// TIA Portal V20 export
// export: Created 2025-12-01T14:56:37.1159273Z, ExportSetting None, DisplayName Totally Integrated Automation Portal, DisplayVersion V20 Update 3, DisplayName TIA Portal Openness, DisplayVersion V20 Update 3, DisplayName TIA Portal Version Control Interface, DisplayVersion V20 Update 3, DisplayName STEP 7 Professional, DisplayVersion V20 Update 3, DisplayName STEP 7 Safety, DisplayVersion V20 Update 2, DisplayName WinCC Basic/Comfort/Advanced, DisplayVersion V20 Update 3, DisplayName WinCC Professional, DisplayVersion V20 Update 3, DisplayName WinCC Unified, DisplayVersion V20 Update 3
FUNCTION_BLOCK "FB12_M_PASO_ELEV_E1E2E3E4_S1S2S3S4_UPDW"   // FB12, LAD
TITLE = Control del Ramal de Salidas
{ S7_Optimized_Access := 'FALSE' }
AUTHOR : M_ELEVA
NAME : 20160509
VERSION : 3.7
// stored: AutoNumber false, SetENOAutomatically false
   VAR_INPUT
      Mesa : UInt;   // Mesa de la FB
      Error_Tx : Bool;   // Error en el Tx
      EnTension : Bool;   // Existe Tension en la Mesa
      Termico_Tx : Bool;   // Proteccion del Tx
      pHsMx_1 : Bool;   // pHs de la Mesa (Para Entrada por E3E4)
      pHsMx_2 : Bool;   // pHs de la Mesa (Para Entrada por E1E2)
      pHsMx_PR1 : Bool;   // pHs de Protrusion de la Mesa. Nota: No existe >> ON
      pHsMx_PR3 : Bool;   // pHs de Protrusion de la Mesa. Nota: No existe >> ON
      Avance_Tx : Bool;   // Avance del Tx
      Retroceso_Tx : Bool;   // Retroceso del Tx
      Termico_MELEV : Bool;   // Protecion de la Mesa Elevadora
      MELEV_DetectorSeg : Bool;   // Detector de Seguridad >>> Mesa Elevadora
      MELEV_UP : Bool;   // Posicion Arriba >>> Mesa Elevadora
      MELEV_DW : Bool;   // Posicion Abajo >>> Mesa Elevadora
      MELEV_EnMovimiento : Bool;   // EnMovimiento >>> Mesa Elevadora
      Pos_Rep_Vacio_DW : Bool;   // Pos. Reposo Vacia DW >>> Config
      Pos_Rep_Vacio_UP : Bool;   // Pos. Reposo Vacia UP >>> Config
      Pos_Rep_Carga_DW : Bool;   // Pos. Reposo Cargada DW >>> Config
      Pos_Rep_Carga_UP : Bool;   // Pos. Reposo Cargada UP >>> Config
      MAnt_DescargaAct_M1_DW : Bool;   // E1 >> Mesa Anterior DescargaAct
      AVTF_Ent_M1_DW : Bool;   // E1 >> Mesa Anterior AVTF
      P_Mens_Ent_M1_DW : Bool;   // E1 >> Mesa Anterior P_Mens
      MAnt_DescargaAct_M3_DW : Bool;   // E3 >> Mesa Anterior DescargaAct
      AVTF_Ent_M3_DW : Bool;   // E3 >> Mesa Anterior AVTF
      P_Mens_Ent_M3_DW : Bool;   // E3 >> Mesa Anterior P_Mens
      PTF_Sal_M1_DW : Bool;   // S1 >> Mesa Siguiente PTF
      FTF_Sal_M1_DW : Bool;   // S1 >> Mesa Siguiente FTF
      PTF_Sal_M3_DW : Bool;   // S3 >> Mesa Siguiente PTF
      FTF_Sal_M3_DW : Bool;   // S3 >> Mesa Siguiente FTF
      MSig_CargaAct_M1_DW : Bool;
      MSig_CargaAct_M3_DW : Bool;
      MAnt_DescargaAct_M2_UP : Bool;   // E2 >> Mesa Anterior DescargaAct
      AVF_Ent_M2_UP : Bool;   // E2 >> Mesa Anterior AVTF
      P_Mens_Ent_M2_UP : Bool;   // E2 >> Mesa Anterior P_Mens
      MAnt_DescargaAct_M4_UP : Bool;   // E4 >> Mesa Anterior DescargaAct
      AVTF_Ent_M4_UP : Bool;   // E4 >> Mesa Anterior AVTF
      P_Mens_Ent_M4_UP : Bool;   // E4 >> Mesa Anterior P_Mens
      PTF_Sal_M2_UP : Bool;   // S2 >> Mesa Siguiente PTF
      FTF_Sal_M2_UP : Bool;   // S2 >> Mesa Siguiente FTF
      PTF_Sal_M4_UP : Bool;   // S4 >> Mesa Siguiente PTF
      FTF_Sal_M4_UP : Bool;   // S4 >> Mesa Siguiente FTF
      MSig_CargaAct_M2_UP : Bool;
      MSig_CargaAct_M4_UP : Bool;
      Mx_VelocidadLenta_In : Bool;   // Forzar a Velociada Lenta
      F_ENV_MENS_Mx : Bool;   // Fin de Envio de Mensaje
      OrdSal_M1_DW : Bool;   // Orden de Salida por S1
      OrdSal_M3_DW : Bool;   // Orden de Salida por S3
      OrdSal_M2_UP : Bool;   // Orden de Salida por S2
      OrdSal_M4_UP : Bool;   // Orden de Salida por S4
      V_CNT_pHsMx : Int := 1000;   // Valor de Presencia
      V_CNT_pHsMx_FTF : Int := 200;   // Valor para activar FTF. Nota: < = V_CNT_pHsMx.
      V_CNTSeg_pHsMx : Int := 2000;   // Valor de Seguriadad para Presencia
      V_CNT_PasoLenta : Int := 2000;   // Valor de Paso a Lenta
      V_CNT_ApHsMx : Int := 200;   // Valor de Ausencia
      V_CNTSeg_ApHsMx : Int := 2000;   // Valor de Seguriadad para Ausencia
      V_TOut_Tx_Mx : Int := 30000;   // TimeOut de Entrada por E1
      V_TOut_MELEV : Int := 5000;   // TimeOut de Mesa Elevadora
      V_TMP_Protrusion : Int := 200;   // TMP de Protrusion
      V_CNT_PerdidapHs : Int := 1000;   // CNT de Perdida de pHs
   END_VAR
   VAR_OUTPUT
      P_EnvMens_PMx : Bool;   // Permiso de Enviar Mensaje de Presencia
      P_RecepOK_Mx : Bool;   // Recepcion OK
      PTF_Ent_M1_DW : Bool;   // E1 >> Mesa Anterior PTF
      FTF_Ent_M1_DW : Bool;   // E1 >> Mesa Anterior FTF
      PTF_Ent_M3_DW : Bool;   // E3 >> Mesa Anterior PTF
      FTF_Ent_M3_DW : Bool;   // E3 >> Mesa Anterior FTF
      AVTF_Sal_M1_DW : Bool;   // S1 >> Mesa Siguiente AVTF
      P_Mens_Sal_M1_DW : Bool;   // S1 >> Mesa Siguiente P_Mens
      AVTF_Sal_M3_DW : Bool;   // S3 >> Mesa Siguiente AVTF
      P_Mens_Sal_M3_DW : Bool;   // S3 >> Mesa Siguiente P_Mens
      PTF_Ent_M2_UP : Bool;   // E2 >> Mesa Anterior PTF
      FTF_Ent_M2_UP : Bool;   // E2 >> Mesa Anterior FTF
      PTF_Ent_M4_UP : Bool;   // E4 >> Mesa Anterior PTF
      FTF_Ent_M4_UP : Bool;   // E4 >> Mesa Anterior FTF
      AVTF_Sal_M2_UP : Bool;   // S2 >> Mesa Siguiente AVTF
      P_Mens_Sal_M2_UP : Bool;   // S2 >> Mesa Siguiente P_Mens
      AVTF_Sal_M4_UP : Bool;   // S4 >> Mesa Siguiente AVTF
      P_Mens_Sal_M4_UP : Bool;   // S4 >> Mesa Siguiente P_Mens
   END_VAR
   VAR
      Anular_pr1 : Bool;   // ???
      Anular_pr3 : Bool;   // ???
      Mx_ET00 : Bool;
      Mx_ET01 { ExternalWritable := 'False'} : Bool;
      Mx_ET02 : Bool;
      Mx_ET08 : Bool;
      Mx_ET09 : Bool;
      Mx_ET10 : Bool;
      Mx_ET11 : Bool;
      Mx_ET12 : Bool;
      Mx_ET110 : Bool;
      Mx_ET111 : Bool;
      Mx_ET50 : Bool;
      Mx_ET51 : Bool;
      Mx_ET150 : Bool;
      Mx_ET151 : Bool;
      Selec_UP : Bool;   // Seleccionado UP de la Mesa Elevadora
      Selec_DW : Bool;   // Seleccionado DW de la Mesa Elevadora
      Selec_M1M2_Entrada : Bool;   // Seleccionado Entrada E1_DW y E2_UP
      Selec_M3M4_Entrada : Bool;   // Seleccionado Entrada E3_DW y E4_UP
      Selec_M1M2_Salida : Bool;   // Seleccionado Salida E1_DW y E2_UP
      Selec_M3M4_Salida : Bool;   // Seleccionado Salida E3_DW y E4_UP
      MEnt_DescargaAct : Bool;   // Interlock >> DesCargaAct de MAnt >> Mx
      AVTF_MEnt : Bool;   // Interlock >> AVTF de MAnt >> Mx
      P_Mens_MEnt : Bool;   // Interlock >> P_Mens de MAnt >> Mx
      PTF_MEnt : Bool;   // Interlock >> PTF de MAnt >> Mx
      FTF_MEnt : Bool;   // Interlock >> FTF de MAnt >> Mx
      AVTF_MSal : Bool;   // Interlock >> AVTF de Mx >> MSig
      P_Mens_MSal : Bool;   // Interlock >> P_Mens de Mx >> MSig
      PTF_MSal : Bool;   // Interlock >> PTF de Mx >> MSig
      FTF_MSal : Bool;   // Interlock >> FTF de Mx >> MSig
      ProtocoloInciado : Bool;   // Iniciado el Envio del Mensaje de Presencia
      STAT_EnvMens_PMx : Bool;   // Interna >> Envio del Mensaje de Presencia
      CNT_pHsMx_FTF_OK : Bool;   // Enviar ya FTF
      CNT_pHsMx { S7_SetPoint := 'True'} : "FB910_CNT_UHS";   // CNT de la Presencia
      CNTSeg_pHsMx { S7_SetPoint := 'True'} : "FB910_CNT_UHS";   // CNT de Seguridad de la Presencia
      CNT_ApHsMx { S7_SetPoint := 'True'} : "FB910_CNT_UHS";   // CNT de la Ausencia
      CNTSeg_ApHsMx { S7_SetPoint := 'True'} : "FB910_CNT_UHS";   // CNT de Seguridad de la Ausencia
      TMP_EnTension { S7_SetPoint := 'True'} : "FB910_CNT_UHS";
      TOut_Av_Mx { S7_SetPoint := 'True'} : "FB910_CNT_UHS";   // Time Out de Entrada de E1 o E2
      TOut_Rt_Mx { S7_SetPoint := 'True'} : "FB910_CNT_UHS";   // Time Out de Entrada de E3 o E4
      TOut_Subir_MELEV { S7_SetPoint := 'True'} : "FB910_CNT_UHS";   // Time Out de Subida de Mesa Elevadora
      TOut_Bajar_MELEV { S7_SetPoint := 'True'} : "FB910_CNT_UHS";   // Time Out de Bajada de Mesa Elevadora
      TMP_Protrusion { S7_SetPoint := 'True'} : "FB910_CNT_UHS";   // TMP de la Protrusion
      CNT_PerdidapHs { S7_SetPoint := 'True'} : "FB910_CNT_UHS";   // CNT de Perdida de pHs
   END_VAR
   VAR_TEMP
      EstadoZona : "EstadoZona";   // Estado de Zona de la Mesa
      EstadoVI : "EstadosMesa";   // Estado del Vehiculo Inteliguente de la Mesa
      ConfigFB : "UDT_ConfigFB";   // Configuracion de la FB de la Mesa
      V_Protrusion : Int;
      Aux_ET00 : Bool;
   END_VAR
   VAR_TEMP   // added for the SCL form of the ladder/FBD networks
      _w1 : Bool;
      _w2 : Bool;
      _w3 : Bool;
      _w4 : Bool;
      _w5 : Bool;
      _w6 : Bool;
   END_VAR
BEGIN

REGION Network 1: INICIALIZAR - Recoger las Variables de Estado de la Mesa
   // Se recoge - Estado_CBx
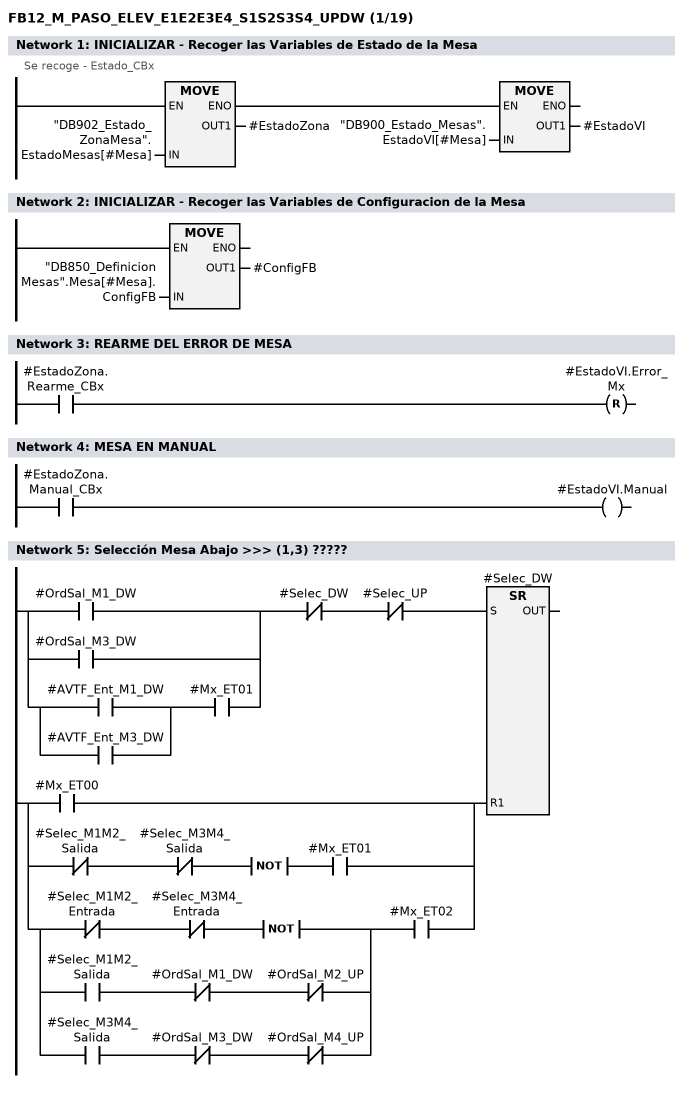
   RUNG wire#powerrail
      Move(in := "DB902_Estado_ZonaMesa".EstadoMesas[#Mesa], out1 => #EstadoZona)
      Move(in := "DB900_Estado_Mesas".EstadoVI[#Mesa], out1 => #EstadoVI)
   END_RUNG
   // the same network as SCL:
   #EstadoZona := "DB902_Estado_ZonaMesa".EstadoMesas[#Mesa];
   #EstadoVI := "DB900_Estado_Mesas".EstadoVI[#Mesa];
END_REGION

REGION Network 2: INICIALIZAR - Recoger las Variables de Configuracion de la Mesa
   RUNG wire#powerrail
      Move(in := "DB850_DefinicionMesas".Mesa[#Mesa].ConfigFB, out1 => #ConfigFB)
   END_RUNG
   // the same network as SCL:
   #ConfigFB := "DB850_DefinicionMesas".Mesa[#Mesa].ConfigFB;
END_REGION

REGION Network 3: REARME DEL ERROR DE MESA
   RUNG wire#powerrail
      Contact( #EstadoZona.Rearme_CBx )
      R_Coil( #EstadoVI.Error_Mx )
   END_RUNG
   // the same network as SCL:
   IF #EstadoZona.Rearme_CBx THEN #EstadoVI.Error_Mx := FALSE; END_IF;
END_REGION

REGION Network 4: MESA EN MANUAL
   RUNG wire#powerrail
      Contact( #EstadoZona.Manual_CBx )
      Coil( #EstadoVI.Manual )
   END_RUNG
   // the same network as SCL:
   #EstadoVI.Manual := #EstadoZona.Manual_CBx;
END_REGION

REGION Network 5: Selección Mesa Abajo >>> (1,3) ?????
   RUNG wire#powerrail
      Contact( #OrdSal_M1_DW )
      wire#w1
      I_Contact( #Selec_DW )
      I_Contact( #Selec_UP )
      S_SR(operand := #Selec_DW, r1 := wire#w4)
   END_RUNG
   RUNG wire#powerrail
      Contact( #OrdSal_M3_DW )
   END_RUNG wire#w1
   RUNG wire#powerrail
      Contact( #AVTF_Ent_M1_DW )
      wire#w2
      Contact( #Mx_ET01 )
   END_RUNG wire#w1
   RUNG wire#powerrail
      Contact( #AVTF_Ent_M3_DW )
   END_RUNG wire#w2
   RUNG wire#powerrail
      Contact( #Mx_ET00 )
   END_RUNG wire#w4
   RUNG wire#powerrail
      I_Contact( #Selec_M1M2_Salida )
      I_Contact( #Selec_M3M4_Salida )
      Not()
      Contact( #Mx_ET01 )
   END_RUNG wire#w4
   RUNG wire#powerrail
      I_Contact( #Selec_M1M2_Entrada )
      I_Contact( #Selec_M3M4_Entrada )
      Not()
      wire#w3
      Contact( #Mx_ET02 )
   END_RUNG wire#w4
   RUNG wire#powerrail
      Contact( #Selec_M1M2_Salida )
      I_Contact( #OrdSal_M1_DW )
      I_Contact( #OrdSal_M2_UP )
   END_RUNG wire#w3
   RUNG wire#powerrail
      Contact( #Selec_M3M4_Salida )
      I_Contact( #OrdSal_M3_DW )
      I_Contact( #OrdSal_M4_UP )
   END_RUNG wire#w3
   // the same network as SCL:
   IF (#OrdSal_M1_DW OR #OrdSal_M3_DW OR ((#AVTF_Ent_M1_DW OR #AVTF_Ent_M3_DW) AND #Mx_ET01)) AND NOT #Selec_DW AND NOT #Selec_UP THEN
       #Selec_DW := TRUE;   // SR flip-flop
   END_IF;
   IF #Mx_ET00 OR (NOT (NOT #Selec_M1M2_Salida AND NOT #Selec_M3M4_Salida) AND #Mx_ET01) OR ((NOT (NOT #Selec_M1M2_Entrada AND NOT #Selec_M3M4_Entrada) OR (#Selec_M1M2_Salida AND NOT #OrdSal_M1_DW AND NOT #OrdSal_M2_UP) OR (#Selec_M3M4_Salida AND NOT #OrdSal_M3_DW AND NOT #OrdSal_M4_UP)) AND #Mx_ET02) THEN
       #Selec_DW := FALSE;
   END_IF;
END_REGION

REGION Network 6: Selección Mesa Arriba >>> (2,4) ?????
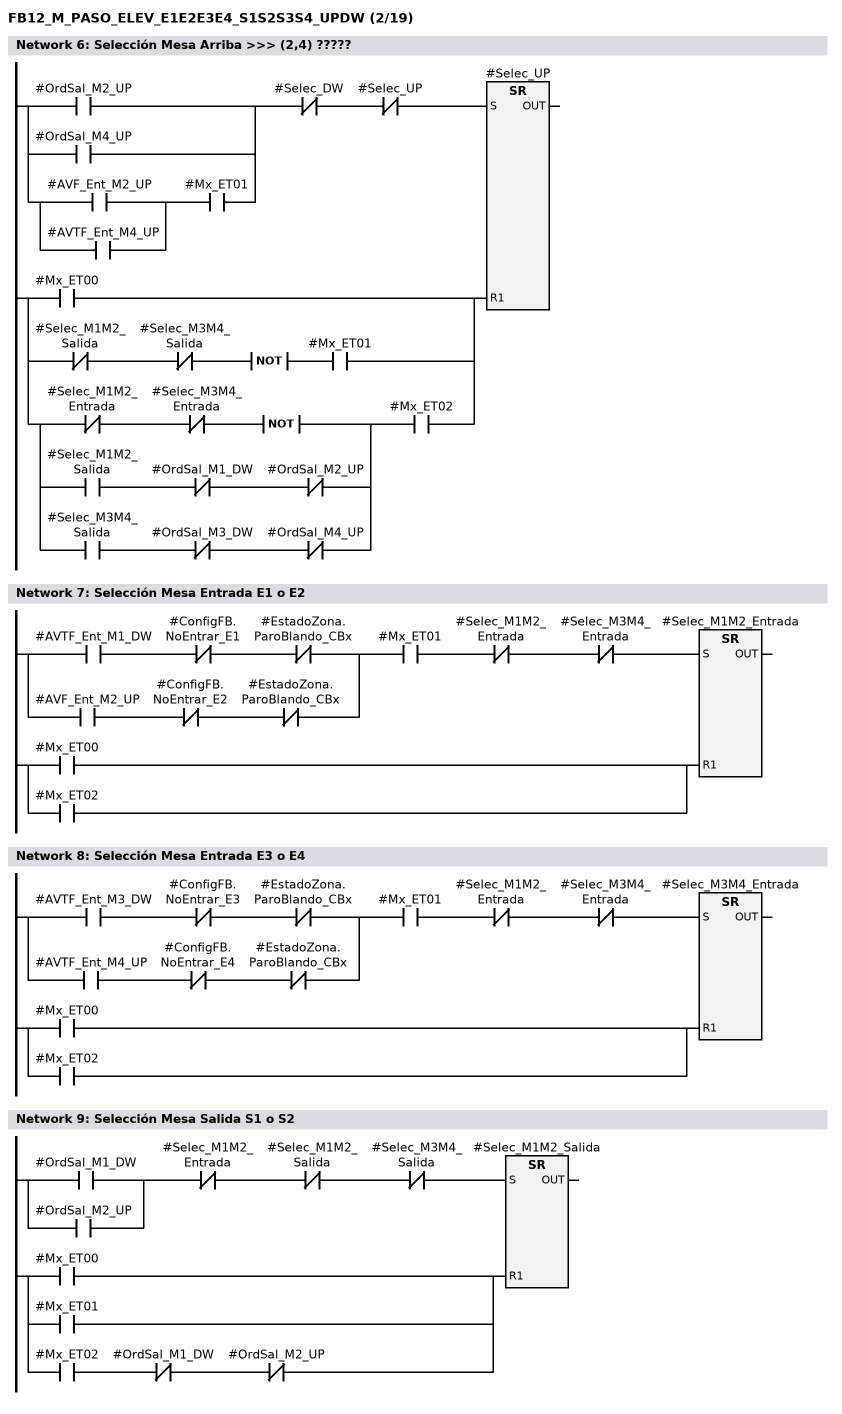
   RUNG wire#powerrail
      Contact( #OrdSal_M2_UP )
      wire#w1
      I_Contact( #Selec_DW )
      I_Contact( #Selec_UP )
      S_SR(operand := #Selec_UP, r1 := wire#w4)
   END_RUNG
   RUNG wire#powerrail
      Contact( #OrdSal_M4_UP )
   END_RUNG wire#w1
   RUNG wire#powerrail
      Contact( #AVF_Ent_M2_UP )
      wire#w2
      Contact( #Mx_ET01 )
   END_RUNG wire#w1
   RUNG wire#powerrail
      Contact( #AVTF_Ent_M4_UP )
   END_RUNG wire#w2
   RUNG wire#powerrail
      Contact( #Mx_ET00 )
   END_RUNG wire#w4
   RUNG wire#powerrail
      I_Contact( #Selec_M1M2_Salida )
      I_Contact( #Selec_M3M4_Salida )
      Not()
      Contact( #Mx_ET01 )
   END_RUNG wire#w4
   RUNG wire#powerrail
      I_Contact( #Selec_M1M2_Entrada )
      I_Contact( #Selec_M3M4_Entrada )
      Not()
      wire#w3
      Contact( #Mx_ET02 )
   END_RUNG wire#w4
   RUNG wire#powerrail
      Contact( #Selec_M1M2_Salida )
      I_Contact( #OrdSal_M1_DW )
      I_Contact( #OrdSal_M2_UP )
   END_RUNG wire#w3
   RUNG wire#powerrail
      Contact( #Selec_M3M4_Salida )
      I_Contact( #OrdSal_M3_DW )
      I_Contact( #OrdSal_M4_UP )
   END_RUNG wire#w3
   // the same network as SCL:
   IF (#OrdSal_M2_UP OR #OrdSal_M4_UP OR ((#AVF_Ent_M2_UP OR #AVTF_Ent_M4_UP) AND #Mx_ET01)) AND NOT #Selec_DW AND NOT #Selec_UP THEN
       #Selec_UP := TRUE;   // SR flip-flop
   END_IF;
   IF #Mx_ET00 OR (NOT (NOT #Selec_M1M2_Salida AND NOT #Selec_M3M4_Salida) AND #Mx_ET01) OR ((NOT (NOT #Selec_M1M2_Entrada AND NOT #Selec_M3M4_Entrada) OR (#Selec_M1M2_Salida AND NOT #OrdSal_M1_DW AND NOT #OrdSal_M2_UP) OR (#Selec_M3M4_Salida AND NOT #OrdSal_M3_DW AND NOT #OrdSal_M4_UP)) AND #Mx_ET02) THEN
       #Selec_UP := FALSE;
   END_IF;
END_REGION

REGION Network 7: Selección Mesa Entrada E1 o E2
   RUNG wire#powerrail
      Contact( #AVTF_Ent_M1_DW )
      I_Contact( #ConfigFB.NoEntrar_E1 )
      I_Contact( #EstadoZona.ParoBlando_CBx )
      wire#w1
      Contact( #Mx_ET01 )
      I_Contact( #Selec_M1M2_Entrada )
      I_Contact( #Selec_M3M4_Entrada )
      S_SR(operand := #Selec_M1M2_Entrada, r1 := wire#w2)
   END_RUNG
   RUNG wire#powerrail
      Contact( #AVF_Ent_M2_UP )
      I_Contact( #ConfigFB.NoEntrar_E2 )
      I_Contact( #EstadoZona.ParoBlando_CBx )
   END_RUNG wire#w1
   RUNG wire#powerrail
      Contact( #Mx_ET00 )
   END_RUNG wire#w2
   RUNG wire#powerrail
      Contact( #Mx_ET02 )
   END_RUNG wire#w2
   // the same network as SCL:
   IF ((#AVTF_Ent_M1_DW AND NOT #ConfigFB.NoEntrar_E1 AND NOT #EstadoZona.ParoBlando_CBx) OR (#AVF_Ent_M2_UP AND NOT #ConfigFB.NoEntrar_E2 AND NOT #EstadoZona.ParoBlando_CBx)) AND #Mx_ET01 AND NOT #Selec_M1M2_Entrada AND NOT #Selec_M3M4_Entrada THEN
       #Selec_M1M2_Entrada := TRUE;   // SR flip-flop
   END_IF;
   IF #Mx_ET00 OR #Mx_ET02 THEN #Selec_M1M2_Entrada := FALSE; END_IF;
END_REGION

REGION Network 8: Selección Mesa Entrada E3 o E4
   RUNG wire#powerrail
      Contact( #AVTF_Ent_M3_DW )
      I_Contact( #ConfigFB.NoEntrar_E3 )
      I_Contact( #EstadoZona.ParoBlando_CBx )
      wire#w1
      Contact( #Mx_ET01 )
      I_Contact( #Selec_M1M2_Entrada )
      I_Contact( #Selec_M3M4_Entrada )
      S_SR(operand := #Selec_M3M4_Entrada, r1 := wire#w2)
   END_RUNG
   RUNG wire#powerrail
      Contact( #AVTF_Ent_M4_UP )
      I_Contact( #ConfigFB.NoEntrar_E4 )
      I_Contact( #EstadoZona.ParoBlando_CBx )
   END_RUNG wire#w1
   RUNG wire#powerrail
      Contact( #Mx_ET00 )
   END_RUNG wire#w2
   RUNG wire#powerrail
      Contact( #Mx_ET02 )
   END_RUNG wire#w2
   // the same network as SCL:
   IF ((#AVTF_Ent_M3_DW AND NOT #ConfigFB.NoEntrar_E3 AND NOT #EstadoZona.ParoBlando_CBx) OR (#AVTF_Ent_M4_UP AND NOT #ConfigFB.NoEntrar_E4 AND NOT #EstadoZona.ParoBlando_CBx)) AND #Mx_ET01 AND NOT #Selec_M1M2_Entrada AND NOT #Selec_M3M4_Entrada THEN
       #Selec_M3M4_Entrada := TRUE;   // SR flip-flop
   END_IF;
   IF #Mx_ET00 OR #Mx_ET02 THEN #Selec_M3M4_Entrada := FALSE; END_IF;
END_REGION

REGION Network 9: Selección Mesa Salida S1 o S2
   RUNG wire#powerrail
      Contact( #OrdSal_M1_DW )
      wire#w1
      I_Contact( #Selec_M1M2_Entrada )
      I_Contact( #Selec_M1M2_Salida )
      I_Contact( #Selec_M3M4_Salida )
      S_SR(operand := #Selec_M1M2_Salida, r1 := wire#w2)
   END_RUNG
   RUNG wire#powerrail
      Contact( #OrdSal_M2_UP )
   END_RUNG wire#w1
   RUNG wire#powerrail
      Contact( #Mx_ET00 )
   END_RUNG wire#w2
   RUNG wire#powerrail
      Contact( #Mx_ET01 )
   END_RUNG wire#w2
   RUNG wire#powerrail
      Contact( #Mx_ET02 )
      I_Contact( #OrdSal_M1_DW )
      I_Contact( #OrdSal_M2_UP )
   END_RUNG wire#w2
   // the same network as SCL:
   IF (#OrdSal_M1_DW OR #OrdSal_M2_UP) AND NOT #Selec_M1M2_Entrada AND NOT #Selec_M1M2_Salida AND NOT #Selec_M3M4_Salida THEN
       #Selec_M1M2_Salida := TRUE;   // SR flip-flop
   END_IF;
   IF #Mx_ET00 OR #Mx_ET01 OR (#Mx_ET02 AND NOT #OrdSal_M1_DW AND NOT #OrdSal_M2_UP) THEN
       #Selec_M1M2_Salida := FALSE;
   END_IF;
END_REGION

REGION Network 10: Selección Mesa Salida S3 o S4
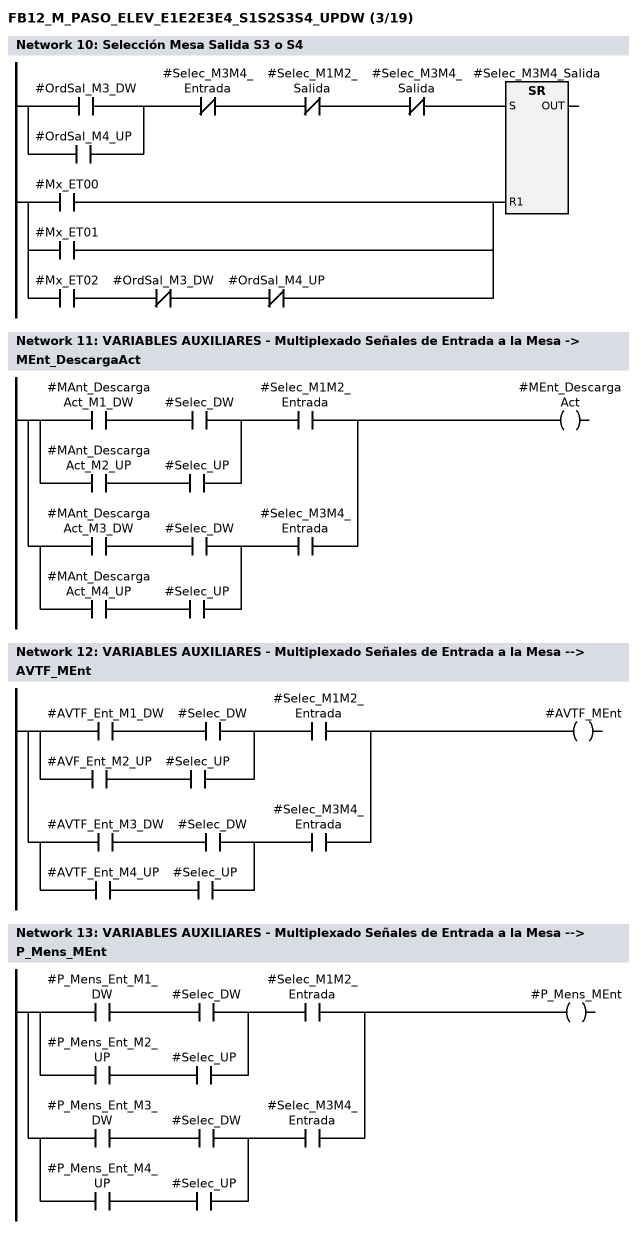
   RUNG wire#powerrail
      Contact( #OrdSal_M3_DW )
      wire#w1
      I_Contact( #Selec_M3M4_Entrada )
      I_Contact( #Selec_M1M2_Salida )
      I_Contact( #Selec_M3M4_Salida )
      S_SR(operand := #Selec_M3M4_Salida, r1 := wire#w2)
   END_RUNG
   RUNG wire#powerrail
      Contact( #OrdSal_M4_UP )
   END_RUNG wire#w1
   RUNG wire#powerrail
      Contact( #Mx_ET00 )
   END_RUNG wire#w2
   RUNG wire#powerrail
      Contact( #Mx_ET01 )
   END_RUNG wire#w2
   RUNG wire#powerrail
      Contact( #Mx_ET02 )
      I_Contact( #OrdSal_M3_DW )
      I_Contact( #OrdSal_M4_UP )
   END_RUNG wire#w2
   // the same network as SCL:
   IF (#OrdSal_M3_DW OR #OrdSal_M4_UP) AND NOT #Selec_M3M4_Entrada AND NOT #Selec_M1M2_Salida AND NOT #Selec_M3M4_Salida THEN
       #Selec_M3M4_Salida := TRUE;   // SR flip-flop
   END_IF;
   IF #Mx_ET00 OR #Mx_ET01 OR (#Mx_ET02 AND NOT #OrdSal_M3_DW AND NOT #OrdSal_M4_UP) THEN
       #Selec_M3M4_Salida := FALSE;
   END_IF;
END_REGION

REGION Network 11: VARIABLES AUXILIARES - Multiplexado Señales de Entrada a la Mesa -> MEnt_DescargaAct
   RUNG wire#powerrail
      Contact( #MAnt_DescargaAct_M1_DW )
      Contact( #Selec_DW )
      wire#w1
      Contact( #Selec_M1M2_Entrada )
      wire#w2
      Coil( #MEnt_DescargaAct )
   END_RUNG
   RUNG wire#powerrail
      Contact( #MAnt_DescargaAct_M2_UP )
      Contact( #Selec_UP )
   END_RUNG wire#w1
   RUNG wire#powerrail
      Contact( #MAnt_DescargaAct_M3_DW )
      Contact( #Selec_DW )
      wire#w3
      Contact( #Selec_M3M4_Entrada )
   END_RUNG wire#w2
   RUNG wire#powerrail
      Contact( #MAnt_DescargaAct_M4_UP )
      Contact( #Selec_UP )
   END_RUNG wire#w3
   // the same network as SCL:
   #MEnt_DescargaAct := (((#MAnt_DescargaAct_M1_DW AND #Selec_DW) OR (#MAnt_DescargaAct_M2_UP AND #Selec_UP)) AND #Selec_M1M2_Entrada) OR (((#MAnt_DescargaAct_M3_DW AND #Selec_DW) OR (#MAnt_DescargaAct_M4_UP AND #Selec_UP)) AND #Selec_M3M4_Entrada);
END_REGION

REGION Network 12: VARIABLES AUXILIARES - Multiplexado Señales de Entrada a la Mesa --> AVTF_MEnt
   RUNG wire#powerrail
      Contact( #AVTF_Ent_M1_DW )
      Contact( #Selec_DW )
      wire#w1
      Contact( #Selec_M1M2_Entrada )
      wire#w2
      Coil( #AVTF_MEnt )
   END_RUNG
   RUNG wire#powerrail
      Contact( #AVF_Ent_M2_UP )
      Contact( #Selec_UP )
   END_RUNG wire#w1
   RUNG wire#powerrail
      Contact( #AVTF_Ent_M3_DW )
      Contact( #Selec_DW )
      wire#w3
      Contact( #Selec_M3M4_Entrada )
   END_RUNG wire#w2
   RUNG wire#powerrail
      Contact( #AVTF_Ent_M4_UP )
      Contact( #Selec_UP )
   END_RUNG wire#w3
   // the same network as SCL:
   #AVTF_MEnt := (((#AVTF_Ent_M1_DW AND #Selec_DW) OR (#AVF_Ent_M2_UP AND #Selec_UP)) AND #Selec_M1M2_Entrada) OR (((#AVTF_Ent_M3_DW AND #Selec_DW) OR (#AVTF_Ent_M4_UP AND #Selec_UP)) AND #Selec_M3M4_Entrada);
END_REGION

REGION Network 13: VARIABLES AUXILIARES - Multiplexado Señales de Entrada a la Mesa --> P_Mens_MEnt
   RUNG wire#powerrail
      Contact( #P_Mens_Ent_M1_DW )
      Contact( #Selec_DW )
      wire#w1
      Contact( #Selec_M1M2_Entrada )
      wire#w2
      Coil( #P_Mens_MEnt )
   END_RUNG
   RUNG wire#powerrail
      Contact( #P_Mens_Ent_M2_UP )
      Contact( #Selec_UP )
   END_RUNG wire#w1
   RUNG wire#powerrail
      Contact( #P_Mens_Ent_M3_DW )
      Contact( #Selec_DW )
      wire#w3
      Contact( #Selec_M3M4_Entrada )
   END_RUNG wire#w2
   RUNG wire#powerrail
      Contact( #P_Mens_Ent_M4_UP )
      Contact( #Selec_UP )
   END_RUNG wire#w3
   // the same network as SCL:
   #P_Mens_MEnt := (((#P_Mens_Ent_M1_DW AND #Selec_DW) OR (#P_Mens_Ent_M2_UP AND #Selec_UP)) AND #Selec_M1M2_Entrada) OR (((#P_Mens_Ent_M3_DW AND #Selec_DW) OR (#P_Mens_Ent_M4_UP AND #Selec_UP)) AND #Selec_M3M4_Entrada);
END_REGION

REGION Network 14: VARIABLES AUXILIARES - Multiplexado Señales de Salida de la Mesa--> PTF_MSal
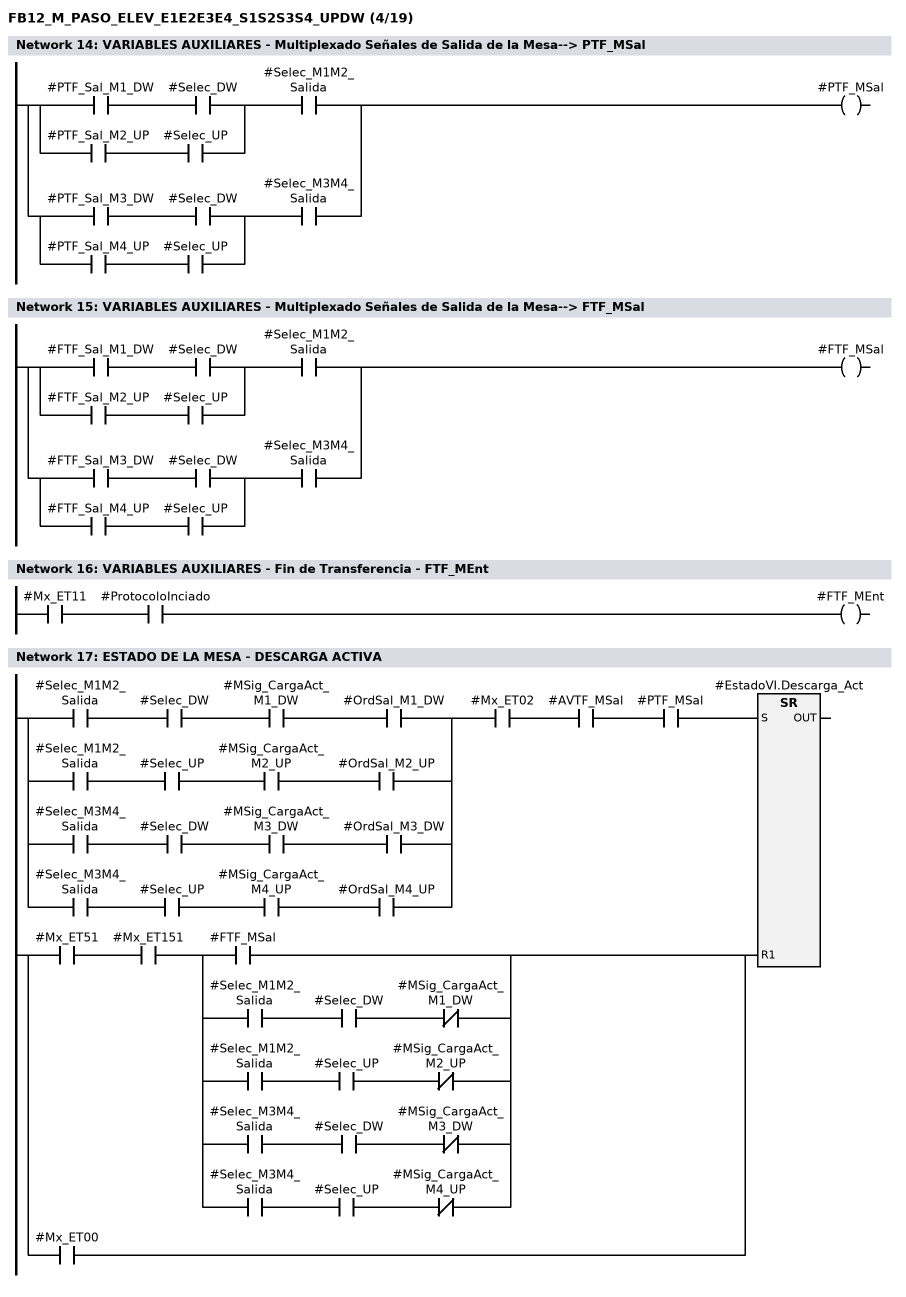
   RUNG wire#powerrail
      Contact( #PTF_Sal_M1_DW )
      Contact( #Selec_DW )
      wire#w1
      Contact( #Selec_M1M2_Salida )
      wire#w2
      Coil( #PTF_MSal )
   END_RUNG
   RUNG wire#powerrail
      Contact( #PTF_Sal_M2_UP )
      Contact( #Selec_UP )
   END_RUNG wire#w1
   RUNG wire#powerrail
      Contact( #PTF_Sal_M3_DW )
      Contact( #Selec_DW )
      wire#w3
      Contact( #Selec_M3M4_Salida )
   END_RUNG wire#w2
   RUNG wire#powerrail
      Contact( #PTF_Sal_M4_UP )
      Contact( #Selec_UP )
   END_RUNG wire#w3
   // the same network as SCL:
   #PTF_MSal := (((#PTF_Sal_M1_DW AND #Selec_DW) OR (#PTF_Sal_M2_UP AND #Selec_UP)) AND #Selec_M1M2_Salida) OR (((#PTF_Sal_M3_DW AND #Selec_DW) OR (#PTF_Sal_M4_UP AND #Selec_UP)) AND #Selec_M3M4_Salida);
END_REGION

REGION Network 15: VARIABLES AUXILIARES - Multiplexado Señales de Salida de la Mesa--> FTF_MSal
   RUNG wire#powerrail
      Contact( #FTF_Sal_M1_DW )
      Contact( #Selec_DW )
      wire#w1
      Contact( #Selec_M1M2_Salida )
      wire#w2
      Coil( #FTF_MSal )
   END_RUNG
   RUNG wire#powerrail
      Contact( #FTF_Sal_M2_UP )
      Contact( #Selec_UP )
   END_RUNG wire#w1
   RUNG wire#powerrail
      Contact( #FTF_Sal_M3_DW )
      Contact( #Selec_DW )
      wire#w3
      Contact( #Selec_M3M4_Salida )
   END_RUNG wire#w2
   RUNG wire#powerrail
      Contact( #FTF_Sal_M4_UP )
      Contact( #Selec_UP )
   END_RUNG wire#w3
   // the same network as SCL:
   #FTF_MSal := (((#FTF_Sal_M1_DW AND #Selec_DW) OR (#FTF_Sal_M2_UP AND #Selec_UP)) AND #Selec_M1M2_Salida) OR (((#FTF_Sal_M3_DW AND #Selec_DW) OR (#FTF_Sal_M4_UP AND #Selec_UP)) AND #Selec_M3M4_Salida);
END_REGION

REGION Network 16: VARIABLES AUXILIARES - Fin de Transferencia - FTF_MEnt
   RUNG wire#powerrail
      Contact( #Mx_ET11 )
      Contact( #ProtocoloInciado )
      Coil( #FTF_MEnt )
   END_RUNG
   // the same network as SCL:
   #FTF_MEnt := #Mx_ET11 AND #ProtocoloInciado;
END_REGION

REGION Network 17: ESTADO DE LA MESA - DESCARGA ACTIVA
   RUNG wire#powerrail
      Contact( #Selec_M1M2_Salida )
      Contact( #Selec_DW )
      Contact( #MSig_CargaAct_M1_DW )
      Contact( #OrdSal_M1_DW )
      wire#w1
      Contact( #Mx_ET02 )
      Contact( #AVTF_MSal )
      Contact( #PTF_MSal )
      S_SR(operand := #EstadoVI.Descarga_Act, r1 := wire#w3)
   END_RUNG
   RUNG wire#powerrail
      Contact( #Selec_M1M2_Salida )
      Contact( #Selec_UP )
      Contact( #MSig_CargaAct_M2_UP )
      Contact( #OrdSal_M2_UP )
   END_RUNG wire#w1
   RUNG wire#powerrail
      Contact( #Selec_M3M4_Salida )
      Contact( #Selec_DW )
      Contact( #MSig_CargaAct_M3_DW )
      Contact( #OrdSal_M3_DW )
   END_RUNG wire#w1
   RUNG wire#powerrail
      Contact( #Selec_M3M4_Salida )
      Contact( #Selec_UP )
      Contact( #MSig_CargaAct_M4_UP )
      Contact( #OrdSal_M4_UP )
   END_RUNG wire#w1
   RUNG wire#powerrail
      Contact( #Mx_ET51 )
      Contact( #Mx_ET151 )
      wire#w2
      Contact( #FTF_MSal )
   END_RUNG wire#w3
   RUNG wire#w2
      Contact( #Selec_M1M2_Salida )
      Contact( #Selec_DW )
      I_Contact( #MSig_CargaAct_M1_DW )
   END_RUNG wire#w3
   RUNG wire#w2
      Contact( #Selec_M1M2_Salida )
      Contact( #Selec_UP )
      I_Contact( #MSig_CargaAct_M2_UP )
   END_RUNG wire#w3
   RUNG wire#w2
      Contact( #Selec_M3M4_Salida )
      Contact( #Selec_DW )
      I_Contact( #MSig_CargaAct_M3_DW )
   END_RUNG wire#w3
   RUNG wire#w2
      Contact( #Selec_M3M4_Salida )
      Contact( #Selec_UP )
      I_Contact( #MSig_CargaAct_M4_UP )
   END_RUNG wire#w3
   RUNG wire#powerrail
      Contact( #Mx_ET00 )
   END_RUNG wire#w3
   // the same network as SCL:
   IF ((#Selec_M1M2_Salida AND #Selec_DW AND #MSig_CargaAct_M1_DW AND #OrdSal_M1_DW) OR (#Selec_M1M2_Salida AND #Selec_UP AND #MSig_CargaAct_M2_UP AND #OrdSal_M2_UP) OR (#Selec_M3M4_Salida AND #Selec_DW AND #MSig_CargaAct_M3_DW AND #OrdSal_M3_DW) OR (#Selec_M3M4_Salida AND #Selec_UP AND #MSig_CargaAct_M4_UP AND #OrdSal_M4_UP)) AND #Mx_ET02 AND #AVTF_MSal AND #PTF_MSal THEN
       #EstadoVI.Descarga_Act := TRUE;   // SR flip-flop
   END_IF;
   IF (#Mx_ET51 AND #Mx_ET151 AND (#FTF_MSal OR (#Selec_M1M2_Salida AND #Selec_DW AND NOT #MSig_CargaAct_M1_DW) OR (#Selec_M1M2_Salida AND #Selec_UP AND NOT #MSig_CargaAct_M2_UP) OR (#Selec_M3M4_Salida AND #Selec_DW AND NOT #MSig_CargaAct_M3_DW) OR (#Selec_M3M4_Salida AND #Selec_UP AND NOT #MSig_CargaAct_M4_UP))) OR #Mx_ET00 THEN
       #EstadoVI.Descarga_Act := FALSE;
   END_IF;
END_REGION

REGION Network 18: ET151 - CONTROL DESCARGA MESA - PROTOCOLO ORDEN
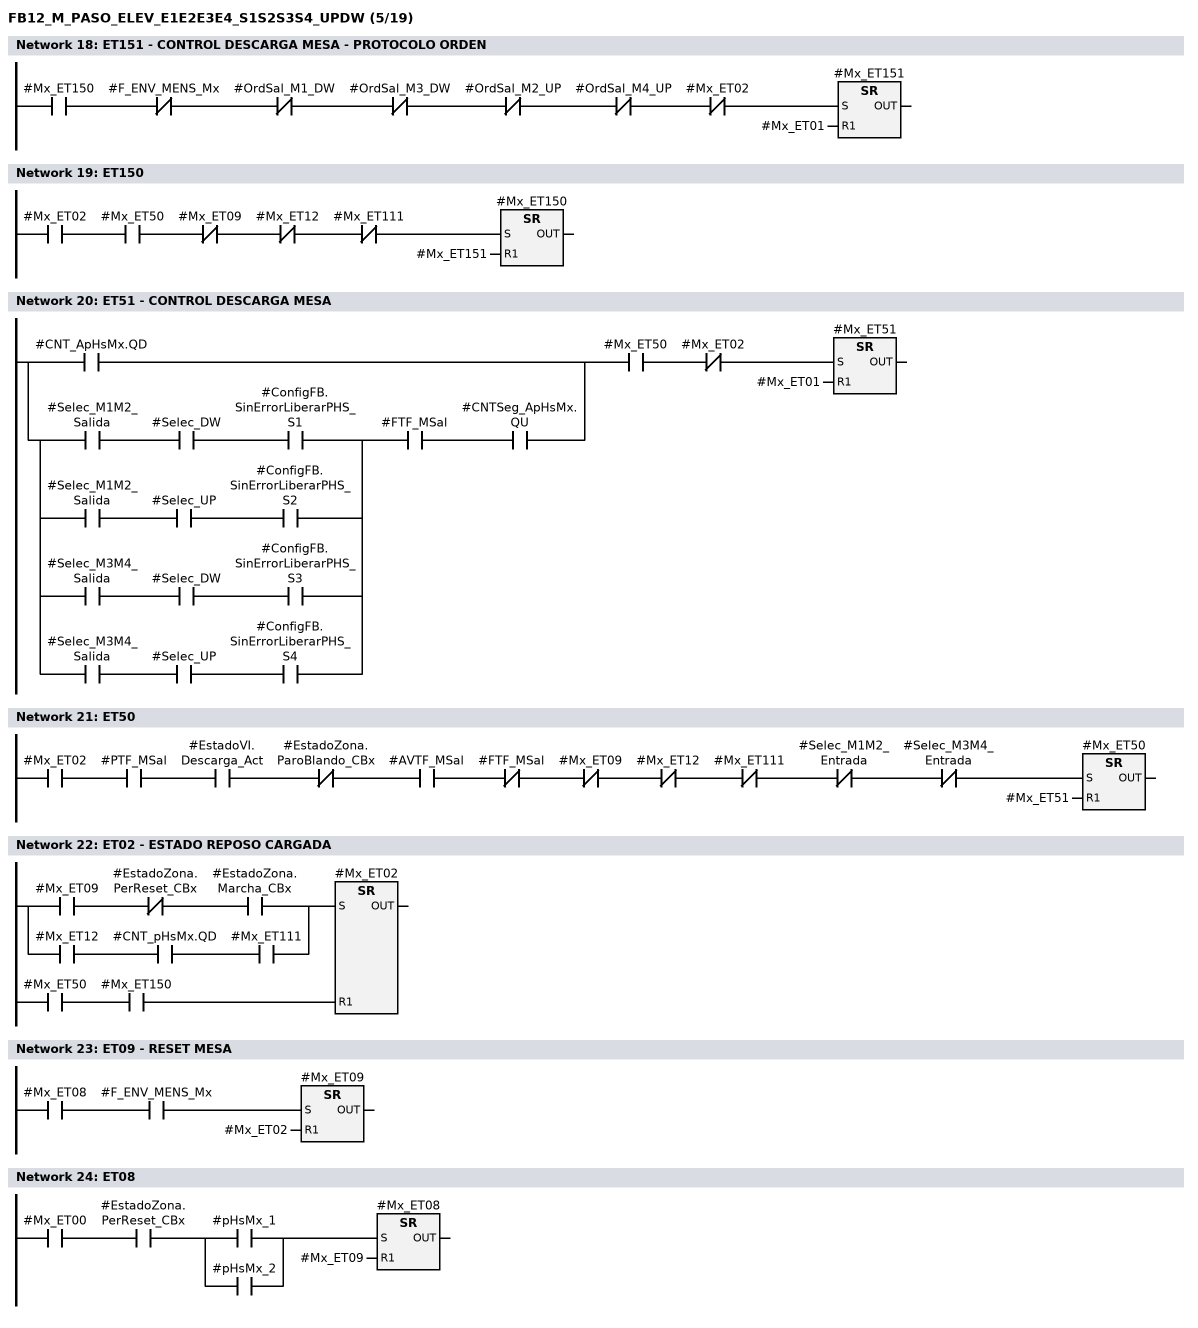
   RUNG wire#powerrail
      Contact( #Mx_ET150 )
      I_Contact( #F_ENV_MENS_Mx )
      I_Contact( #OrdSal_M1_DW )
      I_Contact( #OrdSal_M3_DW )
      I_Contact( #OrdSal_M2_UP )
      I_Contact( #OrdSal_M4_UP )
      I_Contact( #Mx_ET02 )
      S_SR(operand := #Mx_ET151, r1 := #Mx_ET01)
   END_RUNG
   // the same network as SCL:
   IF #Mx_ET150 AND NOT #F_ENV_MENS_Mx AND NOT #OrdSal_M1_DW AND NOT #OrdSal_M3_DW AND NOT #OrdSal_M2_UP AND NOT #OrdSal_M4_UP AND NOT #Mx_ET02 THEN
       #Mx_ET151 := TRUE;   // SR flip-flop
   END_IF;
   IF #Mx_ET01 THEN #Mx_ET151 := FALSE; END_IF;
END_REGION

REGION Network 19: ET150
   RUNG wire#powerrail
      Contact( #Mx_ET02 )
      Contact( #Mx_ET50 )
      I_Contact( #Mx_ET09 )
      I_Contact( #Mx_ET12 )
      I_Contact( #Mx_ET111 )
      S_SR(operand := #Mx_ET150, r1 := #Mx_ET151)
   END_RUNG
   // the same network as SCL:
   IF #Mx_ET02 AND #Mx_ET50 AND NOT #Mx_ET09 AND NOT #Mx_ET12 AND NOT #Mx_ET111 THEN
       #Mx_ET150 := TRUE;   // SR flip-flop
   END_IF;
   IF #Mx_ET151 THEN #Mx_ET150 := FALSE; END_IF;
END_REGION

REGION Network 20: ET51 - CONTROL DESCARGA MESA
   RUNG wire#powerrail
      Contact( #CNT_ApHsMx.QD )
      wire#w1
      Contact( #Mx_ET50 )
      I_Contact( #Mx_ET02 )
      S_SR(operand := #Mx_ET51, r1 := #Mx_ET01)
   END_RUNG
   RUNG wire#powerrail
      Contact( #Selec_M1M2_Salida )
      Contact( #Selec_DW )
      Contact( #ConfigFB.SinErrorLiberarPHS_S1 )
      wire#w2
      Contact( #FTF_MSal )
      Contact( #CNTSeg_ApHsMx.QU )
   END_RUNG wire#w1
   RUNG wire#powerrail
      Contact( #Selec_M1M2_Salida )
      Contact( #Selec_UP )
      Contact( #ConfigFB.SinErrorLiberarPHS_S2 )
   END_RUNG wire#w2
   RUNG wire#powerrail
      Contact( #Selec_M3M4_Salida )
      Contact( #Selec_DW )
      Contact( #ConfigFB.SinErrorLiberarPHS_S3 )
   END_RUNG wire#w2
   RUNG wire#powerrail
      Contact( #Selec_M3M4_Salida )
      Contact( #Selec_UP )
      Contact( #ConfigFB.SinErrorLiberarPHS_S4 )
   END_RUNG wire#w2
   // the same network as SCL:
   IF (#CNT_ApHsMx.QD OR (((#Selec_M1M2_Salida AND #Selec_DW AND #ConfigFB.SinErrorLiberarPHS_S1) OR (#Selec_M1M2_Salida AND #Selec_UP AND #ConfigFB.SinErrorLiberarPHS_S2) OR (#Selec_M3M4_Salida AND #Selec_DW AND #ConfigFB.SinErrorLiberarPHS_S3) OR (#Selec_M3M4_Salida AND #Selec_UP AND #ConfigFB.SinErrorLiberarPHS_S4)) AND #FTF_MSal AND #CNTSeg_ApHsMx.QU)) AND #Mx_ET50 AND NOT #Mx_ET02 THEN
       #Mx_ET51 := TRUE;   // SR flip-flop
   END_IF;
   IF #Mx_ET01 THEN #Mx_ET51 := FALSE; END_IF;
END_REGION

REGION Network 21: ET50
   RUNG wire#powerrail
      Contact( #Mx_ET02 )
      Contact( #PTF_MSal )
      Contact( #EstadoVI.Descarga_Act )
      I_Contact( #EstadoZona.ParoBlando_CBx )
      Contact( #AVTF_MSal )
      I_Contact( #FTF_MSal )
      I_Contact( #Mx_ET09 )
      I_Contact( #Mx_ET12 )
      I_Contact( #Mx_ET111 )
      I_Contact( #Selec_M1M2_Entrada )
      I_Contact( #Selec_M3M4_Entrada )
      S_SR(operand := #Mx_ET50, r1 := #Mx_ET51)
   END_RUNG
   // the same network as SCL:
   IF #Mx_ET02 AND #PTF_MSal AND #EstadoVI.Descarga_Act AND NOT #EstadoZona.ParoBlando_CBx AND #AVTF_MSal AND NOT #FTF_MSal AND NOT #Mx_ET09 AND NOT #Mx_ET12 AND NOT #Mx_ET111 AND NOT #Selec_M1M2_Entrada AND NOT #Selec_M3M4_Entrada THEN
       #Mx_ET50 := TRUE;   // SR flip-flop
   END_IF;
   IF #Mx_ET51 THEN #Mx_ET50 := FALSE; END_IF;
END_REGION

REGION Network 22: ET02 - ESTADO REPOSO CARGADA
   RUNG wire#powerrail
      Contact( #Mx_ET09 )
      I_Contact( #EstadoZona.PerReset_CBx )
      Contact( #EstadoZona.Marcha_CBx )
      wire#w1
      S_SR(operand := #Mx_ET02, r1 := wire#w2)
   END_RUNG
   RUNG wire#powerrail
      Contact( #Mx_ET12 )
      Contact( #CNT_pHsMx.QD )
      Contact( #Mx_ET111 )
   END_RUNG wire#w1
   RUNG wire#powerrail
      Contact( #Mx_ET50 )
      Contact( #Mx_ET150 )
   END_RUNG wire#w2
   // the same network as SCL:
   IF (#Mx_ET09 AND NOT #EstadoZona.PerReset_CBx AND #EstadoZona.Marcha_CBx) OR (#Mx_ET12 AND #CNT_pHsMx.QD AND #Mx_ET111) THEN
       #Mx_ET02 := TRUE;   // SR flip-flop
   END_IF;
   IF #Mx_ET50 AND #Mx_ET150 THEN #Mx_ET02 := FALSE; END_IF;
END_REGION

REGION Network 23: ET09 - RESET MESA
   RUNG wire#powerrail
      Contact( #Mx_ET08 )
      Contact( #F_ENV_MENS_Mx )
      S_SR(operand := #Mx_ET09, r1 := #Mx_ET02)
   END_RUNG
   // the same network as SCL:
   IF #Mx_ET08 AND #F_ENV_MENS_Mx THEN
       #Mx_ET09 := TRUE;   // SR flip-flop
   END_IF;
   IF #Mx_ET02 THEN #Mx_ET09 := FALSE; END_IF;
END_REGION

REGION Network 24: ET08
   RUNG wire#powerrail
      Contact( #Mx_ET00 )
      Contact( #EstadoZona.PerReset_CBx )
      wire#w1
      Contact( #pHsMx_1 )
      wire#w2
      S_SR(operand := #Mx_ET08, r1 := #Mx_ET09)
   END_RUNG
   RUNG wire#w1
      Contact( #pHsMx_2 )
   END_RUNG wire#w2
   // the same network as SCL:
   IF #Mx_ET00 AND #EstadoZona.PerReset_CBx AND (#pHsMx_1 OR #pHsMx_2) THEN
       #Mx_ET08 := TRUE;   // SR flip-flop
   END_IF;
   IF #Mx_ET09 THEN #Mx_ET08 := FALSE; END_IF;
END_REGION

REGION Network 25: ET111 - CONTROL CARGA MESA - MENSAJE DE PRESENCIA
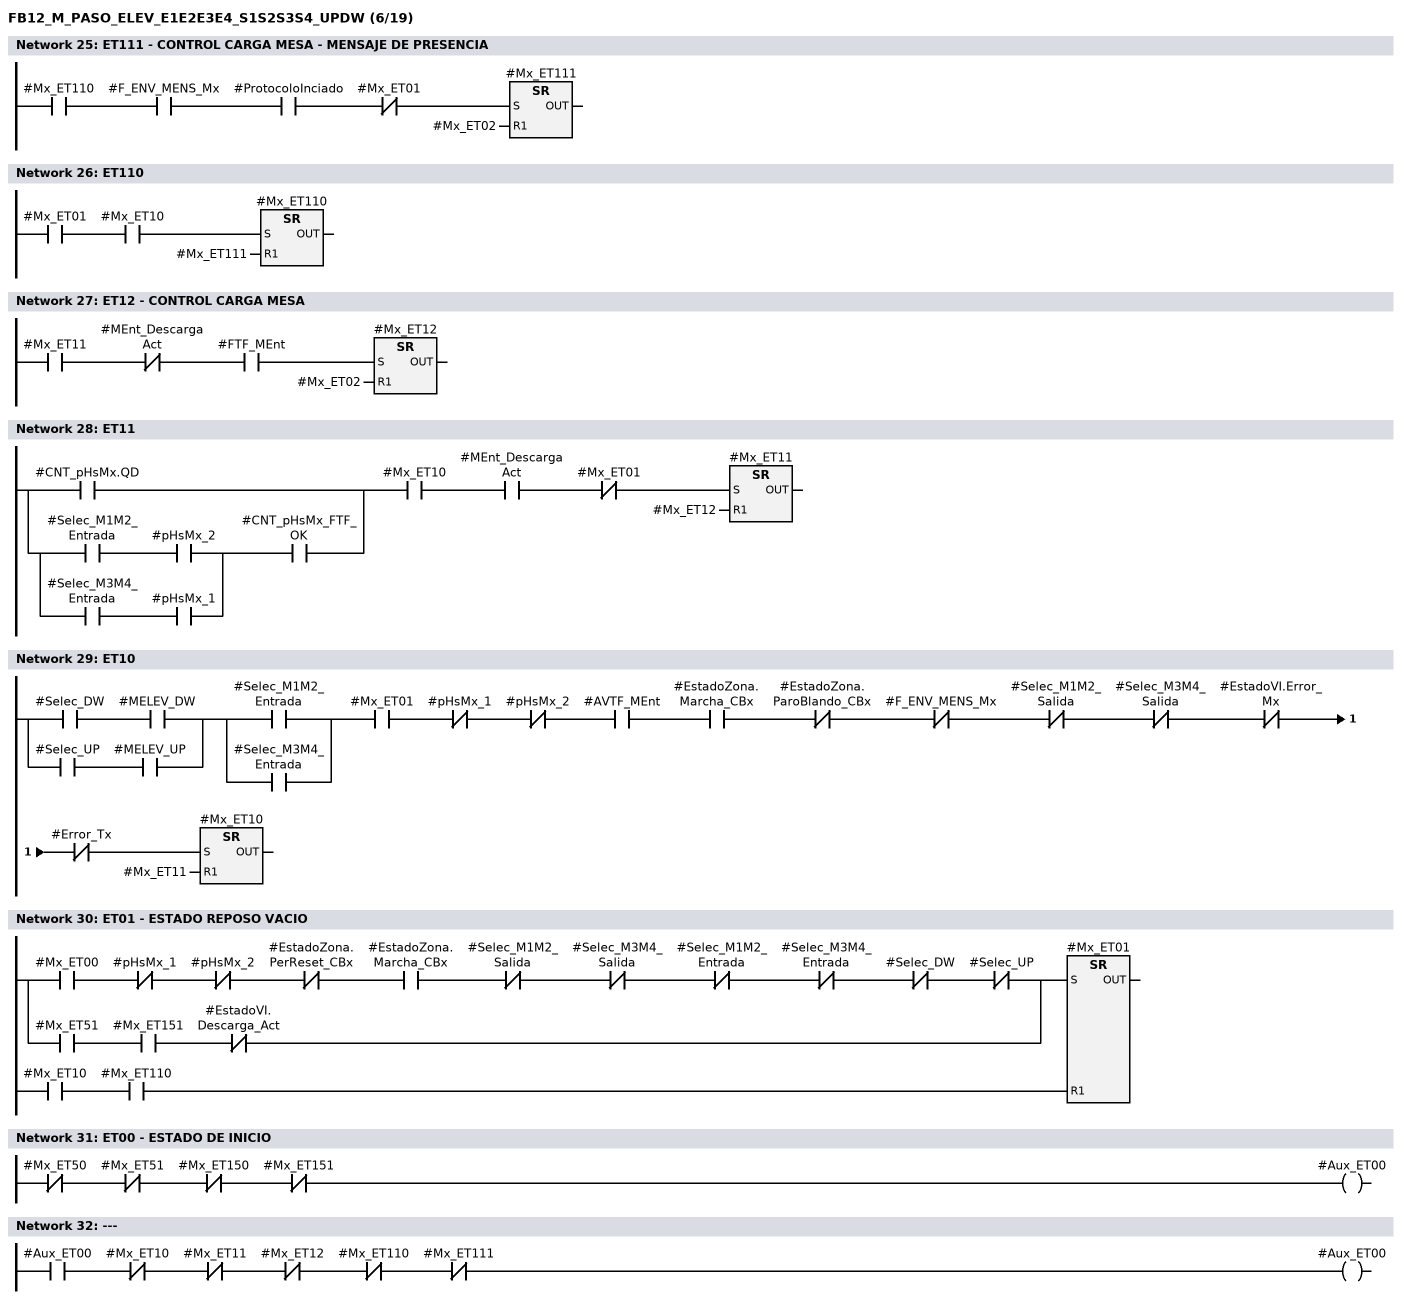
   RUNG wire#powerrail
      Contact( #Mx_ET110 )
      Contact( #F_ENV_MENS_Mx )
      Contact( #ProtocoloInciado )
      I_Contact( #Mx_ET01 )
      S_SR(operand := #Mx_ET111, r1 := #Mx_ET02)
   END_RUNG
   // the same network as SCL:
   IF #Mx_ET110 AND #F_ENV_MENS_Mx AND #ProtocoloInciado AND NOT #Mx_ET01 THEN
       #Mx_ET111 := TRUE;   // SR flip-flop
   END_IF;
   IF #Mx_ET02 THEN #Mx_ET111 := FALSE; END_IF;
END_REGION

REGION Network 26: ET110
   RUNG wire#powerrail
      Contact( #Mx_ET01 )
      Contact( #Mx_ET10 )
      S_SR(operand := #Mx_ET110, r1 := #Mx_ET111)
   END_RUNG
   // the same network as SCL:
   IF #Mx_ET01 AND #Mx_ET10 THEN
       #Mx_ET110 := TRUE;   // SR flip-flop
   END_IF;
   IF #Mx_ET111 THEN #Mx_ET110 := FALSE; END_IF;
END_REGION

REGION Network 27: ET12 - CONTROL CARGA MESA
   RUNG wire#powerrail
      Contact( #Mx_ET11 )
      I_Contact( #MEnt_DescargaAct )
      Contact( #FTF_MEnt )
      S_SR(operand := #Mx_ET12, r1 := #Mx_ET02)
   END_RUNG
   // the same network as SCL:
   IF #Mx_ET11 AND NOT #MEnt_DescargaAct AND #FTF_MEnt THEN
       #Mx_ET12 := TRUE;   // SR flip-flop
   END_IF;
   IF #Mx_ET02 THEN #Mx_ET12 := FALSE; END_IF;
END_REGION

REGION Network 28: ET11
   RUNG wire#powerrail
      Contact( #CNT_pHsMx.QD )
      wire#w1
      Contact( #Mx_ET10 )
      Contact( #MEnt_DescargaAct )
      I_Contact( #Mx_ET01 )
      S_SR(operand := #Mx_ET11, r1 := #Mx_ET12)
   END_RUNG
   RUNG wire#powerrail
      Contact( #Selec_M1M2_Entrada )
      Contact( #pHsMx_2 )
      wire#w2
      Contact( #CNT_pHsMx_FTF_OK )
   END_RUNG wire#w1
   RUNG wire#powerrail
      Contact( #Selec_M3M4_Entrada )
      Contact( #pHsMx_1 )
   END_RUNG wire#w2
   // the same network as SCL:
   IF (#CNT_pHsMx.QD OR (((#Selec_M1M2_Entrada AND #pHsMx_2) OR (#Selec_M3M4_Entrada AND #pHsMx_1)) AND #CNT_pHsMx_FTF_OK)) AND #Mx_ET10 AND #MEnt_DescargaAct AND NOT #Mx_ET01 THEN
       #Mx_ET11 := TRUE;   // SR flip-flop
   END_IF;
   IF #Mx_ET12 THEN #Mx_ET11 := FALSE; END_IF;
END_REGION

REGION Network 29: ET10
   RUNG wire#powerrail
      Contact( #Selec_DW )
      Contact( #MELEV_DW )
      wire#w1
      Contact( #Selec_M1M2_Entrada )
      wire#w2
      Contact( #Mx_ET01 )
      I_Contact( #pHsMx_1 )
      I_Contact( #pHsMx_2 )
      Contact( #AVTF_MEnt )
      Contact( #EstadoZona.Marcha_CBx )
      I_Contact( #EstadoZona.ParoBlando_CBx )
      I_Contact( #F_ENV_MENS_Mx )
      I_Contact( #Selec_M1M2_Salida )
      I_Contact( #Selec_M3M4_Salida )
      I_Contact( #EstadoVI.Error_Mx )
      I_Contact( #Error_Tx )
      S_SR(operand := #Mx_ET10, r1 := #Mx_ET11)
   END_RUNG
   RUNG wire#powerrail
      Contact( #Selec_UP )
      Contact( #MELEV_UP )
   END_RUNG wire#w1
   RUNG wire#w1
      Contact( #Selec_M3M4_Entrada )
   END_RUNG wire#w2
   // the same network as SCL:
   IF ((#Selec_DW AND #MELEV_DW) OR (#Selec_UP AND #MELEV_UP)) AND (#Selec_M1M2_Entrada OR #Selec_M3M4_Entrada) AND #Mx_ET01 AND NOT #pHsMx_1 AND NOT #pHsMx_2 AND #AVTF_MEnt AND #EstadoZona.Marcha_CBx AND NOT #EstadoZona.ParoBlando_CBx AND NOT #F_ENV_MENS_Mx AND NOT #Selec_M1M2_Salida AND NOT #Selec_M3M4_Salida AND NOT #EstadoVI.Error_Mx AND NOT #Error_Tx THEN
       #Mx_ET10 := TRUE;   // SR flip-flop
   END_IF;
   IF #Mx_ET11 THEN #Mx_ET10 := FALSE; END_IF;
END_REGION

REGION Network 30: ET01 - ESTADO REPOSO VACIO
   RUNG wire#powerrail
      Contact( #Mx_ET00 )
      I_Contact( #pHsMx_1 )
      I_Contact( #pHsMx_2 )
      I_Contact( #EstadoZona.PerReset_CBx )
      Contact( #EstadoZona.Marcha_CBx )
      I_Contact( #Selec_M1M2_Salida )
      I_Contact( #Selec_M3M4_Salida )
      I_Contact( #Selec_M1M2_Entrada )
      I_Contact( #Selec_M3M4_Entrada )
      I_Contact( #Selec_DW )
      I_Contact( #Selec_UP )
      wire#w1
      S_SR(operand := #Mx_ET01, r1 := wire#w2)
   END_RUNG
   RUNG wire#powerrail
      Contact( #Mx_ET51 )
      Contact( #Mx_ET151 )
      I_Contact( #EstadoVI.Descarga_Act )
   END_RUNG wire#w1
   RUNG wire#powerrail
      Contact( #Mx_ET10 )
      Contact( #Mx_ET110 )
   END_RUNG wire#w2
   // the same network as SCL:
   IF (#Mx_ET00 AND NOT #pHsMx_1 AND NOT #pHsMx_2 AND NOT #EstadoZona.PerReset_CBx AND #EstadoZona.Marcha_CBx AND NOT #Selec_M1M2_Salida AND NOT #Selec_M3M4_Salida AND NOT #Selec_M1M2_Entrada AND NOT #Selec_M3M4_Entrada AND NOT #Selec_DW AND NOT #Selec_UP) OR (#Mx_ET51 AND #Mx_ET151 AND NOT #EstadoVI.Descarga_Act) THEN
       #Mx_ET01 := TRUE;   // SR flip-flop
   END_IF;
   IF #Mx_ET10 AND #Mx_ET110 THEN #Mx_ET01 := FALSE; END_IF;
END_REGION

REGION Network 31: ET00 - ESTADO DE INICIO
   RUNG wire#powerrail
      I_Contact( #Mx_ET50 )
      I_Contact( #Mx_ET51 )
      I_Contact( #Mx_ET150 )
      I_Contact( #Mx_ET151 )
      Coil( #Aux_ET00 )
   END_RUNG
   // the same network as SCL:
   #Aux_ET00 := NOT #Mx_ET50 AND NOT #Mx_ET51 AND NOT #Mx_ET150 AND NOT #Mx_ET151;
END_REGION

REGION Network 32: ---
   RUNG wire#powerrail
      Contact( #Aux_ET00 )
      I_Contact( #Mx_ET10 )
      I_Contact( #Mx_ET11 )
      I_Contact( #Mx_ET12 )
      I_Contact( #Mx_ET110 )
      I_Contact( #Mx_ET111 )
      Coil( #Aux_ET00 )
   END_RUNG
   // the same network as SCL:
   #Aux_ET00 := #Aux_ET00 AND NOT #Mx_ET10 AND NOT #Mx_ET11 AND NOT #Mx_ET12 AND NOT #Mx_ET110 AND NOT #Mx_ET111;
END_REGION

REGION Network 33: ---
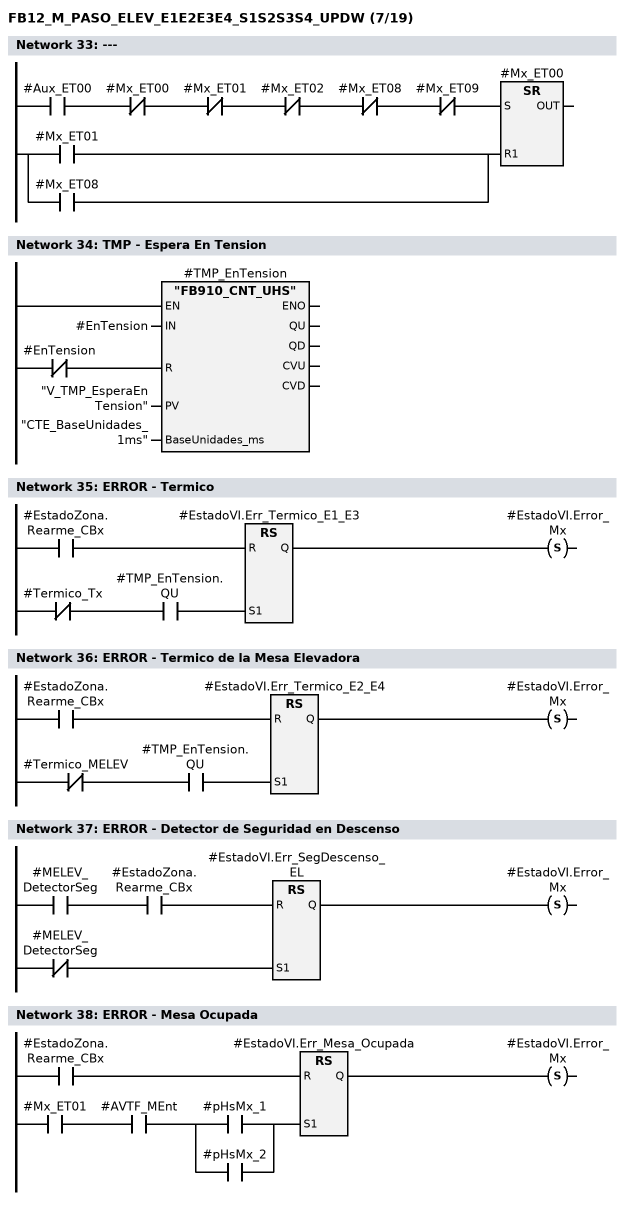
   RUNG wire#powerrail
      Contact( #Aux_ET00 )
      I_Contact( #Mx_ET00 )
      I_Contact( #Mx_ET01 )
      I_Contact( #Mx_ET02 )
      I_Contact( #Mx_ET08 )
      I_Contact( #Mx_ET09 )
      S_SR(operand := #Mx_ET00, r1 := wire#w1)
   END_RUNG
   RUNG wire#powerrail
      Contact( #Mx_ET01 )
   END_RUNG wire#w1
   RUNG wire#powerrail
      Contact( #Mx_ET08 )
   END_RUNG wire#w1
   // the same network as SCL:
   IF #Aux_ET00 AND NOT #Mx_ET00 AND NOT #Mx_ET01 AND NOT #Mx_ET02 AND NOT #Mx_ET08 AND NOT #Mx_ET09 THEN
       #Mx_ET00 := TRUE;   // SR flip-flop
   END_IF;
   IF #Mx_ET01 OR #Mx_ET08 THEN #Mx_ET00 := FALSE; END_IF;
END_REGION

REGION Network 34: TMP - Espera En Tension
   RUNG wire#powerrail
      #TMP_EnTension(R := wire#w1, IN := #EnTension, PV := "V_TMP_EsperaEnTension", BaseUnidades_ms := "CTE_BaseUnidades_1ms", QU =>, QD =>, CVU =>, CVD =>)
   END_RUNG
   RUNG wire#powerrail
      I_Contact( #EnTension )
   END_RUNG wire#w1
   // the same network as SCL:
   #TMP_EnTension(IN := #EnTension,   // "FB910_CNT_UHS"
                  R := NOT #EnTension,
                  PV := "V_TMP_EsperaEnTension",
                  BaseUnidades_ms := "CTE_BaseUnidades_1ms");
END_REGION

REGION Network 35: ERROR - Termico
   RUNG wire#powerrail
      Contact( #EstadoZona.Rearme_CBx )
      S_RS(operand := #EstadoVI.Err_Termico_E1_E3, s1 := wire#w1)
      S_Coil( #EstadoVI.Error_Mx )
   END_RUNG
   RUNG wire#powerrail
      I_Contact( #Termico_Tx )
      Contact( #TMP_EnTension.QU )
   END_RUNG wire#w1
   // the same network as SCL:
   IF #EstadoZona.Rearme_CBx THEN
       #EstadoVI.Err_Termico_E1_E3 := FALSE;   // RS flip-flop
   END_IF;
   IF NOT #Termico_Tx AND #TMP_EnTension.QU THEN #EstadoVI.Err_Termico_E1_E3 := TRUE; END_IF;
   IF #EstadoVI.Err_Termico_E1_E3 THEN #EstadoVI.Error_Mx := TRUE; END_IF;
END_REGION

REGION Network 36: ERROR - Termico de la Mesa Elevadora
   RUNG wire#powerrail
      Contact( #EstadoZona.Rearme_CBx )
      S_RS(operand := #EstadoVI.Err_Termico_E2_E4, s1 := wire#w1)
      S_Coil( #EstadoVI.Error_Mx )
   END_RUNG
   RUNG wire#powerrail
      I_Contact( #Termico_MELEV )
      Contact( #TMP_EnTension.QU )
   END_RUNG wire#w1
   // the same network as SCL:
   IF #EstadoZona.Rearme_CBx THEN
       #EstadoVI.Err_Termico_E2_E4 := FALSE;   // RS flip-flop
   END_IF;
   IF NOT #Termico_MELEV AND #TMP_EnTension.QU THEN #EstadoVI.Err_Termico_E2_E4 := TRUE; END_IF;
   IF #EstadoVI.Err_Termico_E2_E4 THEN #EstadoVI.Error_Mx := TRUE; END_IF;
END_REGION

REGION Network 37: ERROR - Detector de Seguridad en Descenso
   RUNG wire#powerrail
      Contact( #MELEV_DetectorSeg )
      Contact( #EstadoZona.Rearme_CBx )
      S_RS(operand := #EstadoVI.Err_SegDescenso_EL, s1 := wire#w1)
      S_Coil( #EstadoVI.Error_Mx )
   END_RUNG
   RUNG wire#powerrail
      I_Contact( #MELEV_DetectorSeg )
   END_RUNG wire#w1
   // the same network as SCL:
   IF #MELEV_DetectorSeg AND #EstadoZona.Rearme_CBx THEN
       #EstadoVI.Err_SegDescenso_EL := FALSE;   // RS flip-flop
   END_IF;
   IF NOT #MELEV_DetectorSeg THEN #EstadoVI.Err_SegDescenso_EL := TRUE; END_IF;
   IF #EstadoVI.Err_SegDescenso_EL THEN #EstadoVI.Error_Mx := TRUE; END_IF;
END_REGION

REGION Network 38: ERROR - Mesa Ocupada
   RUNG wire#powerrail
      Contact( #EstadoZona.Rearme_CBx )
      S_RS(operand := #EstadoVI.Err_Mesa_Ocupada, s1 := wire#w2)
      S_Coil( #EstadoVI.Error_Mx )
   END_RUNG
   RUNG wire#powerrail
      Contact( #Mx_ET01 )
      Contact( #AVTF_MEnt )
      wire#w1
      Contact( #pHsMx_1 )
   END_RUNG wire#w2
   RUNG wire#w1
      Contact( #pHsMx_2 )
   END_RUNG wire#w2
   // the same network as SCL:
   IF #EstadoZona.Rearme_CBx THEN
       #EstadoVI.Err_Mesa_Ocupada := FALSE;   // RS flip-flop
   END_IF;
   IF #Mx_ET01 AND #AVTF_MEnt AND (#pHsMx_1 OR #pHsMx_2) THEN #EstadoVI.Err_Mesa_Ocupada := TRUE; END_IF;
   IF #EstadoVI.Err_Mesa_Ocupada THEN #EstadoVI.Error_Mx := TRUE; END_IF;
END_REGION

REGION Network 39: CNT - ERROR - Arrastre
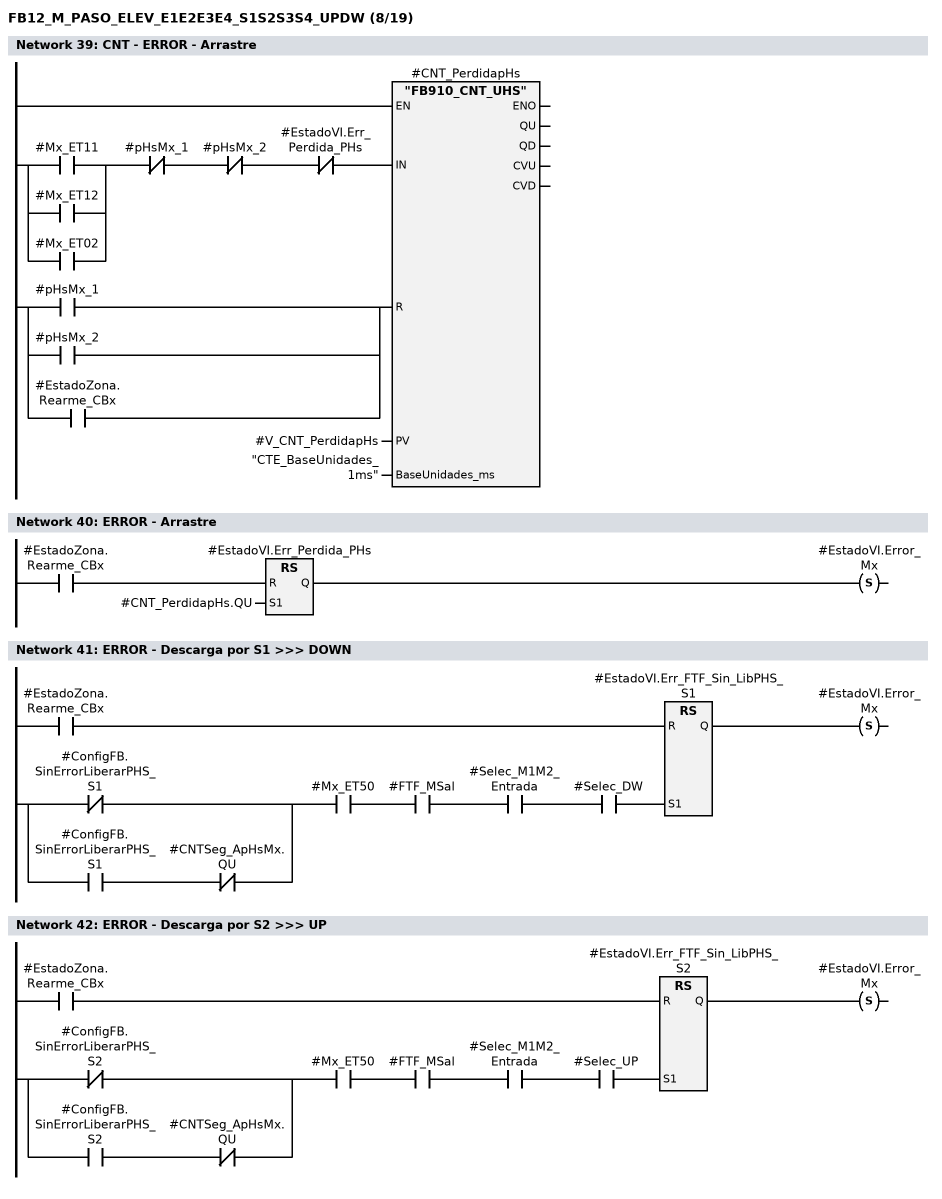
   RUNG wire#powerrail
      #CNT_PerdidapHs(IN := wire#w2, R := wire#w3, PV := #V_CNT_PerdidapHs, BaseUnidades_ms := "CTE_BaseUnidades_1ms", QU =>, QD =>, CVU =>, CVD =>)
   END_RUNG
   RUNG wire#powerrail
      Contact( #Mx_ET11 )
      wire#w1
      I_Contact( #pHsMx_1 )
      I_Contact( #pHsMx_2 )
      I_Contact( #EstadoVI.Err_Perdida_PHs )
   END_RUNG wire#w2
   RUNG wire#powerrail
      Contact( #Mx_ET12 )
   END_RUNG wire#w1
   RUNG wire#powerrail
      Contact( #Mx_ET02 )
   END_RUNG wire#w1
   RUNG wire#powerrail
      Contact( #pHsMx_1 )
   END_RUNG wire#w3
   RUNG wire#powerrail
      Contact( #pHsMx_2 )
   END_RUNG wire#w3
   RUNG wire#powerrail
      Contact( #EstadoZona.Rearme_CBx )
   END_RUNG wire#w3
   // the same network as SCL:
   #CNT_PerdidapHs(IN := (#Mx_ET11 OR #Mx_ET12 OR #Mx_ET02) AND NOT #pHsMx_1 AND NOT #pHsMx_2 AND NOT #EstadoVI.Err_Perdida_PHs,   // "FB910_CNT_UHS"
                   R := #pHsMx_1 OR #pHsMx_2 OR #EstadoZona.Rearme_CBx,
                   PV := #V_CNT_PerdidapHs,
                   BaseUnidades_ms := "CTE_BaseUnidades_1ms");
END_REGION

REGION Network 40: ERROR - Arrastre
   RUNG wire#powerrail
      Contact( #EstadoZona.Rearme_CBx )
      S_RS(operand := #EstadoVI.Err_Perdida_PHs, s1 := #CNT_PerdidapHs.QU)
      S_Coil( #EstadoVI.Error_Mx )
   END_RUNG
   // the same network as SCL:
   IF #EstadoZona.Rearme_CBx THEN
       #EstadoVI.Err_Perdida_PHs := FALSE;   // RS flip-flop
   END_IF;
   IF #CNT_PerdidapHs.QU THEN #EstadoVI.Err_Perdida_PHs := TRUE; END_IF;
   IF #EstadoVI.Err_Perdida_PHs THEN #EstadoVI.Error_Mx := TRUE; END_IF;
END_REGION

REGION Network 41: ERROR - Descarga por S1 >>> DOWN
   RUNG wire#powerrail
      Contact( #EstadoZona.Rearme_CBx )
      S_RS(operand := #EstadoVI.Err_FTF_Sin_LibPHS_S1, s1 := wire#w2)
      S_Coil( #EstadoVI.Error_Mx )
   END_RUNG
   RUNG wire#powerrail
      I_Contact( #ConfigFB.SinErrorLiberarPHS_S1 )
      wire#w1
      Contact( #Mx_ET50 )
      Contact( #FTF_MSal )
      Contact( #Selec_M1M2_Entrada )
      Contact( #Selec_DW )
   END_RUNG wire#w2
   RUNG wire#powerrail
      Contact( #ConfigFB.SinErrorLiberarPHS_S1 )
      I_Contact( #CNTSeg_ApHsMx.QU )
   END_RUNG wire#w1
   // the same network as SCL:
   IF #EstadoZona.Rearme_CBx THEN
       #EstadoVI.Err_FTF_Sin_LibPHS_S1 := FALSE;   // RS flip-flop
   END_IF;
   IF (NOT #ConfigFB.SinErrorLiberarPHS_S1 OR (#ConfigFB.SinErrorLiberarPHS_S1 AND NOT #CNTSeg_ApHsMx.QU)) AND #Mx_ET50 AND #FTF_MSal AND #Selec_M1M2_Entrada AND #Selec_DW THEN
       #EstadoVI.Err_FTF_Sin_LibPHS_S1 := TRUE;
   END_IF;
   IF #EstadoVI.Err_FTF_Sin_LibPHS_S1 THEN #EstadoVI.Error_Mx := TRUE; END_IF;
END_REGION

REGION Network 42: ERROR - Descarga por S2 >>> UP
   RUNG wire#powerrail
      Contact( #EstadoZona.Rearme_CBx )
      S_RS(operand := #EstadoVI.Err_FTF_Sin_LibPHS_S2, s1 := wire#w2)
      S_Coil( #EstadoVI.Error_Mx )
   END_RUNG
   RUNG wire#powerrail
      I_Contact( #ConfigFB.SinErrorLiberarPHS_S2 )
      wire#w1
      Contact( #Mx_ET50 )
      Contact( #FTF_MSal )
      Contact( #Selec_M1M2_Entrada )
      Contact( #Selec_UP )
   END_RUNG wire#w2
   RUNG wire#powerrail
      Contact( #ConfigFB.SinErrorLiberarPHS_S2 )
      I_Contact( #CNTSeg_ApHsMx.QU )
   END_RUNG wire#w1
   // the same network as SCL:
   IF #EstadoZona.Rearme_CBx THEN
       #EstadoVI.Err_FTF_Sin_LibPHS_S2 := FALSE;   // RS flip-flop
   END_IF;
   IF (NOT #ConfigFB.SinErrorLiberarPHS_S2 OR (#ConfigFB.SinErrorLiberarPHS_S2 AND NOT #CNTSeg_ApHsMx.QU)) AND #Mx_ET50 AND #FTF_MSal AND #Selec_M1M2_Entrada AND #Selec_UP THEN
       #EstadoVI.Err_FTF_Sin_LibPHS_S2 := TRUE;
   END_IF;
   IF #EstadoVI.Err_FTF_Sin_LibPHS_S2 THEN #EstadoVI.Error_Mx := TRUE; END_IF;
END_REGION

REGION Network 43: ERROR - Descarga por S3 >>> DOWN
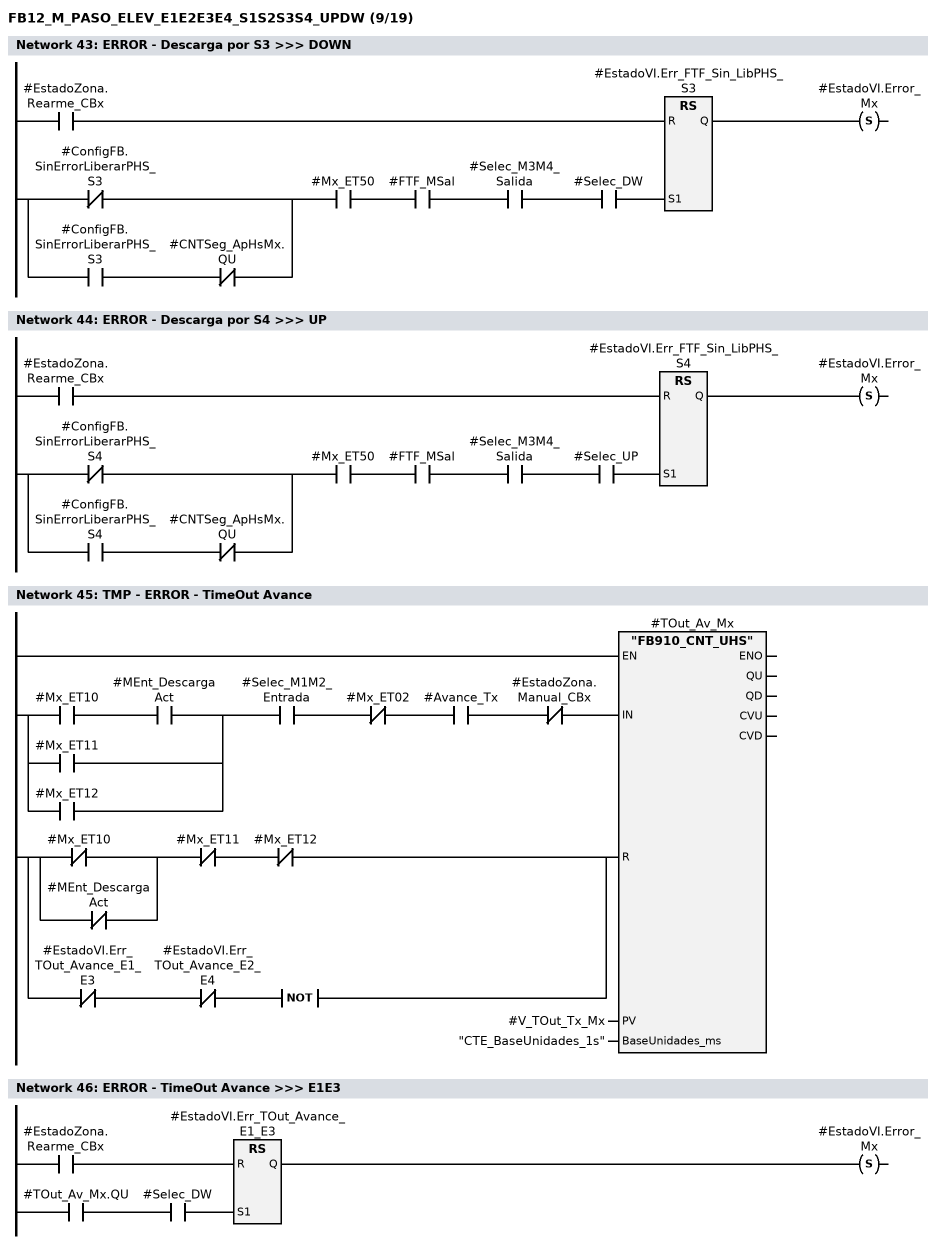
   RUNG wire#powerrail
      Contact( #EstadoZona.Rearme_CBx )
      S_RS(operand := #EstadoVI.Err_FTF_Sin_LibPHS_S3, s1 := wire#w2)
      S_Coil( #EstadoVI.Error_Mx )
   END_RUNG
   RUNG wire#powerrail
      I_Contact( #ConfigFB.SinErrorLiberarPHS_S3 )
      wire#w1
      Contact( #Mx_ET50 )
      Contact( #FTF_MSal )
      Contact( #Selec_M3M4_Salida )
      Contact( #Selec_DW )
   END_RUNG wire#w2
   RUNG wire#powerrail
      Contact( #ConfigFB.SinErrorLiberarPHS_S3 )
      I_Contact( #CNTSeg_ApHsMx.QU )
   END_RUNG wire#w1
   // the same network as SCL:
   IF #EstadoZona.Rearme_CBx THEN
       #EstadoVI.Err_FTF_Sin_LibPHS_S3 := FALSE;   // RS flip-flop
   END_IF;
   IF (NOT #ConfigFB.SinErrorLiberarPHS_S3 OR (#ConfigFB.SinErrorLiberarPHS_S3 AND NOT #CNTSeg_ApHsMx.QU)) AND #Mx_ET50 AND #FTF_MSal AND #Selec_M3M4_Salida AND #Selec_DW THEN
       #EstadoVI.Err_FTF_Sin_LibPHS_S3 := TRUE;
   END_IF;
   IF #EstadoVI.Err_FTF_Sin_LibPHS_S3 THEN #EstadoVI.Error_Mx := TRUE; END_IF;
END_REGION

REGION Network 44: ERROR - Descarga por S4 >>> UP
   RUNG wire#powerrail
      Contact( #EstadoZona.Rearme_CBx )
      S_RS(operand := #EstadoVI.Err_FTF_Sin_LibPHS_S4, s1 := wire#w2)
      S_Coil( #EstadoVI.Error_Mx )
   END_RUNG
   RUNG wire#powerrail
      I_Contact( #ConfigFB.SinErrorLiberarPHS_S4 )
      wire#w1
      Contact( #Mx_ET50 )
      Contact( #FTF_MSal )
      Contact( #Selec_M3M4_Salida )
      Contact( #Selec_UP )
   END_RUNG wire#w2
   RUNG wire#powerrail
      Contact( #ConfigFB.SinErrorLiberarPHS_S4 )
      I_Contact( #CNTSeg_ApHsMx.QU )
   END_RUNG wire#w1
   // the same network as SCL:
   IF #EstadoZona.Rearme_CBx THEN
       #EstadoVI.Err_FTF_Sin_LibPHS_S4 := FALSE;   // RS flip-flop
   END_IF;
   IF (NOT #ConfigFB.SinErrorLiberarPHS_S4 OR (#ConfigFB.SinErrorLiberarPHS_S4 AND NOT #CNTSeg_ApHsMx.QU)) AND #Mx_ET50 AND #FTF_MSal AND #Selec_M3M4_Salida AND #Selec_UP THEN
       #EstadoVI.Err_FTF_Sin_LibPHS_S4 := TRUE;
   END_IF;
   IF #EstadoVI.Err_FTF_Sin_LibPHS_S4 THEN #EstadoVI.Error_Mx := TRUE; END_IF;
END_REGION

REGION Network 45: TMP - ERROR - TimeOut Avance
   RUNG wire#powerrail
      #TOut_Av_Mx(IN := wire#w2, R := wire#w4, PV := #V_TOut_Tx_Mx, BaseUnidades_ms := "CTE_BaseUnidades_1s", QU =>, QD =>, CVU =>, CVD =>)
   END_RUNG
   RUNG wire#powerrail
      Contact( #Mx_ET10 )
      Contact( #MEnt_DescargaAct )
      wire#w1
      Contact( #Selec_M1M2_Entrada )
      I_Contact( #Mx_ET02 )
      Contact( #Avance_Tx )
      I_Contact( #EstadoZona.Manual_CBx )
   END_RUNG wire#w2
   RUNG wire#powerrail
      Contact( #Mx_ET11 )
   END_RUNG wire#w1
   RUNG wire#powerrail
      Contact( #Mx_ET12 )
   END_RUNG wire#w1
   RUNG wire#powerrail
      I_Contact( #Mx_ET10 )
      wire#w3
      I_Contact( #Mx_ET11 )
      I_Contact( #Mx_ET12 )
   END_RUNG wire#w4
   RUNG wire#powerrail
      I_Contact( #MEnt_DescargaAct )
   END_RUNG wire#w3
   RUNG wire#powerrail
      I_Contact( #EstadoVI.Err_TOut_Avance_E1_E3 )
      I_Contact( #EstadoVI.Err_TOut_Avance_E2_E4 )
      Not()
   END_RUNG wire#w4
   // the same network as SCL:
   #TOut_Av_Mx(IN := ((#Mx_ET10 AND #MEnt_DescargaAct) OR #Mx_ET11 OR #Mx_ET12) AND #Selec_M1M2_Entrada AND NOT #Mx_ET02 AND #Avance_Tx AND NOT #EstadoZona.Manual_CBx,   // "FB910_CNT_UHS"
               R := ((NOT #Mx_ET10 OR NOT #MEnt_DescargaAct) AND NOT #Mx_ET11 AND NOT #Mx_ET12) OR NOT (NOT #EstadoVI.Err_TOut_Avance_E1_E3 AND NOT #EstadoVI.Err_TOut_Avance_E2_E4),
               PV := #V_TOut_Tx_Mx,
               BaseUnidades_ms := "CTE_BaseUnidades_1s");
END_REGION

REGION Network 46: ERROR - TimeOut Avance >>> E1E3
   RUNG wire#powerrail
      Contact( #EstadoZona.Rearme_CBx )
      S_RS(operand := #EstadoVI.Err_TOut_Avance_E1_E3, s1 := wire#w1)
      S_Coil( #EstadoVI.Error_Mx )
   END_RUNG
   RUNG wire#powerrail
      Contact( #TOut_Av_Mx.QU )
      Contact( #Selec_DW )
   END_RUNG wire#w1
   // the same network as SCL:
   IF #EstadoZona.Rearme_CBx THEN
       #EstadoVI.Err_TOut_Avance_E1_E3 := FALSE;   // RS flip-flop
   END_IF;
   IF #TOut_Av_Mx.QU AND #Selec_DW THEN #EstadoVI.Err_TOut_Avance_E1_E3 := TRUE; END_IF;
   IF #EstadoVI.Err_TOut_Avance_E1_E3 THEN #EstadoVI.Error_Mx := TRUE; END_IF;
END_REGION

REGION Network 47: ERROR - TimeOut Avance >>> E2E4
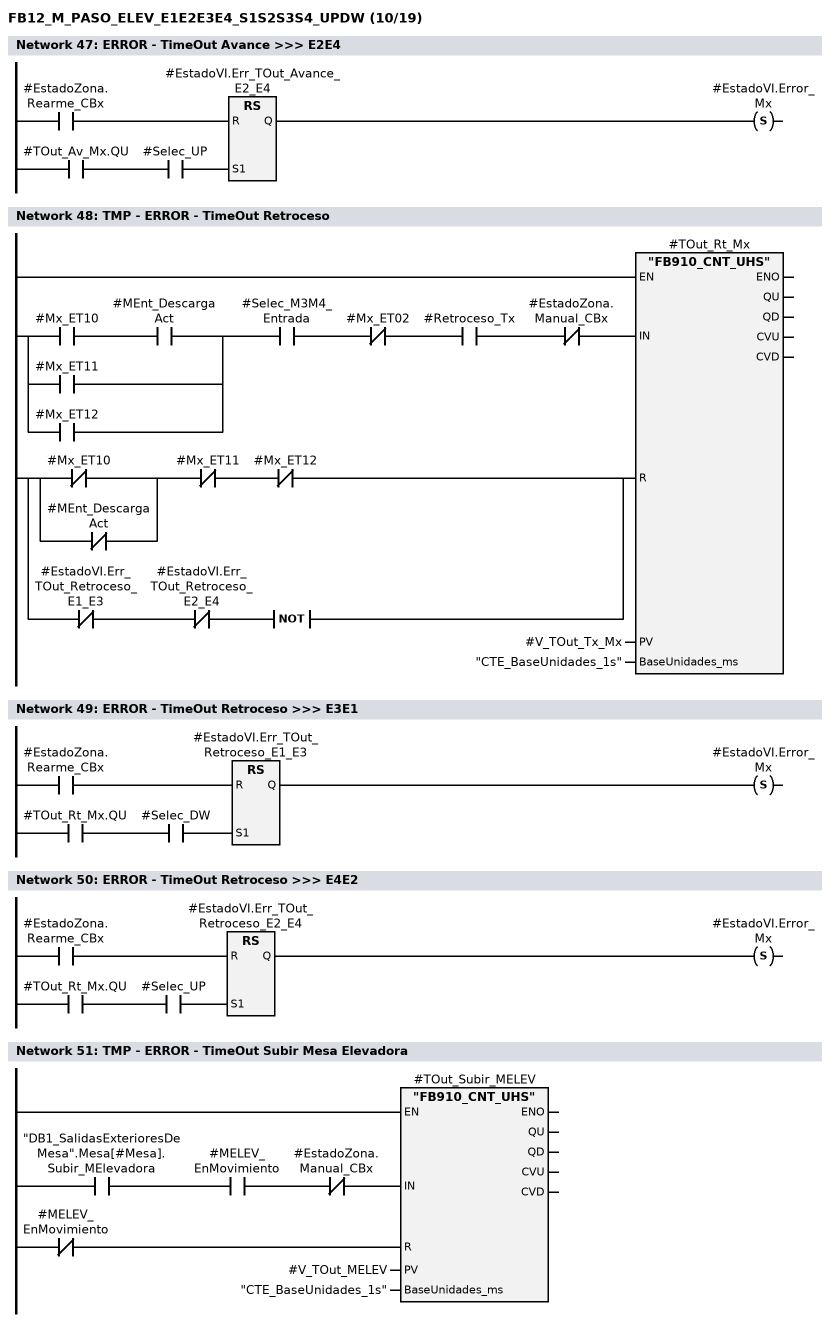
   RUNG wire#powerrail
      Contact( #EstadoZona.Rearme_CBx )
      S_RS(operand := #EstadoVI.Err_TOut_Avance_E2_E4, s1 := wire#w1)
      S_Coil( #EstadoVI.Error_Mx )
   END_RUNG
   RUNG wire#powerrail
      Contact( #TOut_Av_Mx.QU )
      Contact( #Selec_UP )
   END_RUNG wire#w1
   // the same network as SCL:
   IF #EstadoZona.Rearme_CBx THEN
       #EstadoVI.Err_TOut_Avance_E2_E4 := FALSE;   // RS flip-flop
   END_IF;
   IF #TOut_Av_Mx.QU AND #Selec_UP THEN #EstadoVI.Err_TOut_Avance_E2_E4 := TRUE; END_IF;
   IF #EstadoVI.Err_TOut_Avance_E2_E4 THEN #EstadoVI.Error_Mx := TRUE; END_IF;
END_REGION

REGION Network 48: TMP - ERROR - TimeOut Retroceso
   RUNG wire#powerrail
      #TOut_Rt_Mx(IN := wire#w2, R := wire#w4, PV := #V_TOut_Tx_Mx, BaseUnidades_ms := "CTE_BaseUnidades_1s", QU =>, QD =>, CVU =>, CVD =>)
   END_RUNG
   RUNG wire#powerrail
      Contact( #Mx_ET10 )
      Contact( #MEnt_DescargaAct )
      wire#w1
      Contact( #Selec_M3M4_Entrada )
      I_Contact( #Mx_ET02 )
      Contact( #Retroceso_Tx )
      I_Contact( #EstadoZona.Manual_CBx )
   END_RUNG wire#w2
   RUNG wire#powerrail
      Contact( #Mx_ET11 )
   END_RUNG wire#w1
   RUNG wire#powerrail
      Contact( #Mx_ET12 )
   END_RUNG wire#w1
   RUNG wire#powerrail
      I_Contact( #Mx_ET10 )
      wire#w3
      I_Contact( #Mx_ET11 )
      I_Contact( #Mx_ET12 )
   END_RUNG wire#w4
   RUNG wire#powerrail
      I_Contact( #MEnt_DescargaAct )
   END_RUNG wire#w3
   RUNG wire#powerrail
      I_Contact( #EstadoVI.Err_TOut_Retroceso_E1_E3 )
      I_Contact( #EstadoVI.Err_TOut_Retroceso_E2_E4 )
      Not()
   END_RUNG wire#w4
   // the same network as SCL:
   #TOut_Rt_Mx(IN := ((#Mx_ET10 AND #MEnt_DescargaAct) OR #Mx_ET11 OR #Mx_ET12) AND #Selec_M3M4_Entrada AND NOT #Mx_ET02 AND #Retroceso_Tx AND NOT #EstadoZona.Manual_CBx,   // "FB910_CNT_UHS"
               R := ((NOT #Mx_ET10 OR NOT #MEnt_DescargaAct) AND NOT #Mx_ET11 AND NOT #Mx_ET12) OR NOT (NOT #EstadoVI.Err_TOut_Retroceso_E1_E3 AND NOT #EstadoVI.Err_TOut_Retroceso_E2_E4),
               PV := #V_TOut_Tx_Mx,
               BaseUnidades_ms := "CTE_BaseUnidades_1s");
END_REGION

REGION Network 49: ERROR - TimeOut Retroceso >>> E3E1
   RUNG wire#powerrail
      Contact( #EstadoZona.Rearme_CBx )
      S_RS(operand := #EstadoVI.Err_TOut_Retroceso_E1_E3, s1 := wire#w1)
      S_Coil( #EstadoVI.Error_Mx )
   END_RUNG
   RUNG wire#powerrail
      Contact( #TOut_Rt_Mx.QU )
      Contact( #Selec_DW )
   END_RUNG wire#w1
   // the same network as SCL:
   IF #EstadoZona.Rearme_CBx THEN
       #EstadoVI.Err_TOut_Retroceso_E1_E3 := FALSE;   // RS flip-flop
   END_IF;
   IF #TOut_Rt_Mx.QU AND #Selec_DW THEN #EstadoVI.Err_TOut_Retroceso_E1_E3 := TRUE; END_IF;
   IF #EstadoVI.Err_TOut_Retroceso_E1_E3 THEN #EstadoVI.Error_Mx := TRUE; END_IF;
END_REGION

REGION Network 50: ERROR - TimeOut Retroceso >>> E4E2
   RUNG wire#powerrail
      Contact( #EstadoZona.Rearme_CBx )
      S_RS(operand := #EstadoVI.Err_TOut_Retroceso_E2_E4, s1 := wire#w1)
      S_Coil( #EstadoVI.Error_Mx )
   END_RUNG
   RUNG wire#powerrail
      Contact( #TOut_Rt_Mx.QU )
      Contact( #Selec_UP )
   END_RUNG wire#w1
   // the same network as SCL:
   IF #EstadoZona.Rearme_CBx THEN
       #EstadoVI.Err_TOut_Retroceso_E2_E4 := FALSE;   // RS flip-flop
   END_IF;
   IF #TOut_Rt_Mx.QU AND #Selec_UP THEN #EstadoVI.Err_TOut_Retroceso_E2_E4 := TRUE; END_IF;
   IF #EstadoVI.Err_TOut_Retroceso_E2_E4 THEN #EstadoVI.Error_Mx := TRUE; END_IF;
END_REGION

REGION Network 51: TMP - ERROR - TimeOut Subir Mesa Elevadora
   RUNG wire#powerrail
      #TOut_Subir_MELEV(IN := wire#w1, R := wire#w2, PV := #V_TOut_MELEV, BaseUnidades_ms := "CTE_BaseUnidades_1s", QU =>, QD =>, CVU =>, CVD =>)
   END_RUNG
   RUNG wire#powerrail
      Contact( "DB1_SalidasExterioresDeMesa".Mesa[#Mesa].Subir_MElevadora )
      Contact( #MELEV_EnMovimiento )
      I_Contact( #EstadoZona.Manual_CBx )
   END_RUNG wire#w1
   RUNG wire#powerrail
      I_Contact( #MELEV_EnMovimiento )
   END_RUNG wire#w2
   // the same network as SCL:
   #TOut_Subir_MELEV(IN := "DB1_SalidasExterioresDeMesa".Mesa[#Mesa].Subir_MElevadora AND #MELEV_EnMovimiento AND NOT #EstadoZona.Manual_CBx,   // "FB910_CNT_UHS"
                     R := NOT #MELEV_EnMovimiento,
                     PV := #V_TOut_MELEV,
                     BaseUnidades_ms := "CTE_BaseUnidades_1s");
END_REGION

REGION Network 52: ERROR - TimeOut Subir Mesa Elevadora
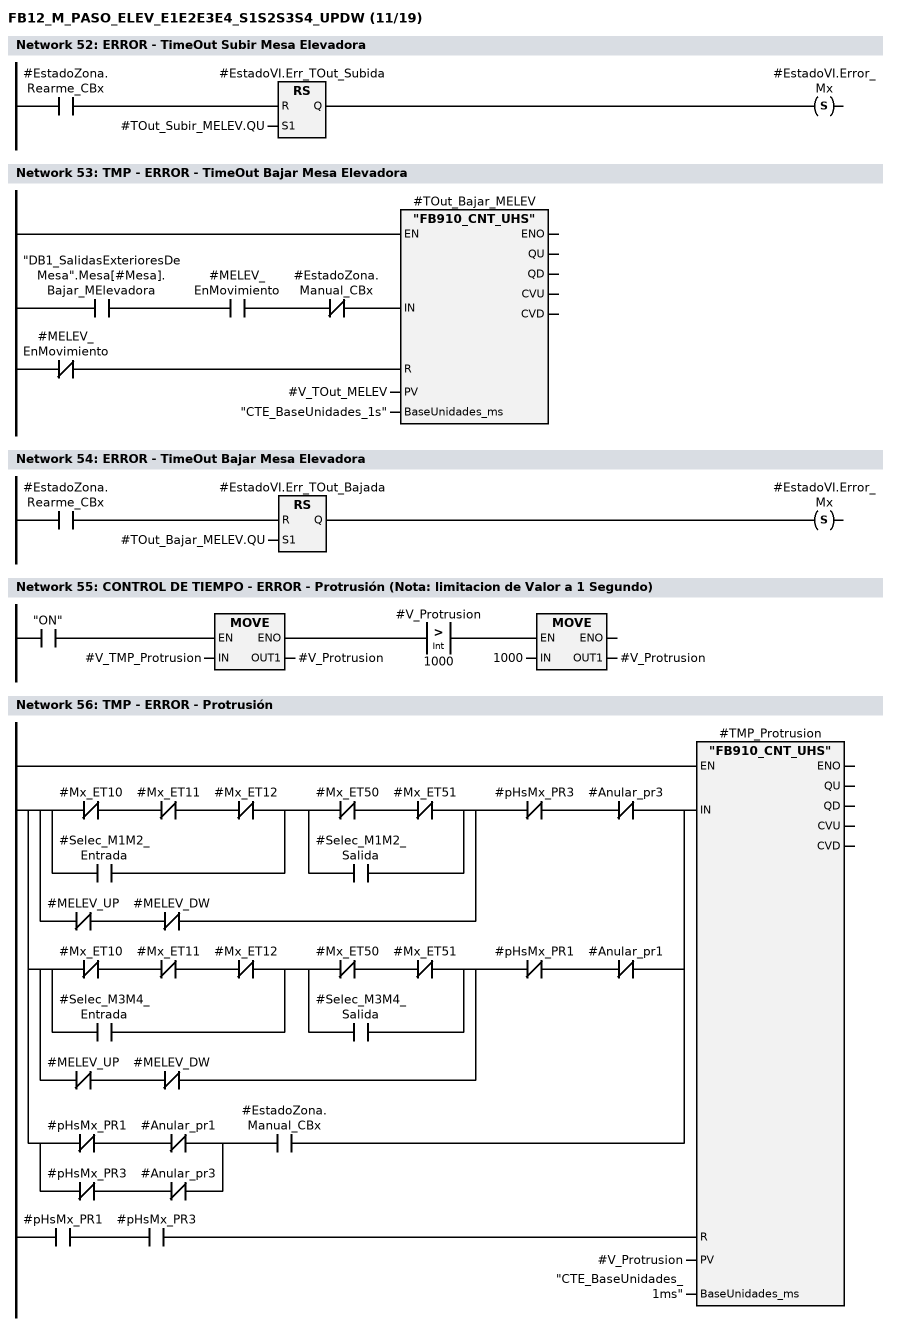
   RUNG wire#powerrail
      Contact( #EstadoZona.Rearme_CBx )
      S_RS(operand := #EstadoVI.Err_TOut_Subida, s1 := #TOut_Subir_MELEV.QU)
      S_Coil( #EstadoVI.Error_Mx )
   END_RUNG
   // the same network as SCL:
   IF #EstadoZona.Rearme_CBx THEN
       #EstadoVI.Err_TOut_Subida := FALSE;   // RS flip-flop
   END_IF;
   IF #TOut_Subir_MELEV.QU THEN #EstadoVI.Err_TOut_Subida := TRUE; END_IF;
   IF #EstadoVI.Err_TOut_Subida THEN #EstadoVI.Error_Mx := TRUE; END_IF;
END_REGION

REGION Network 53: TMP - ERROR - TimeOut Bajar Mesa Elevadora
   RUNG wire#powerrail
      #TOut_Bajar_MELEV(IN := wire#w1, R := wire#w2, PV := #V_TOut_MELEV, BaseUnidades_ms := "CTE_BaseUnidades_1s", QU =>, QD =>, CVU =>, CVD =>)
   END_RUNG
   RUNG wire#powerrail
      Contact( "DB1_SalidasExterioresDeMesa".Mesa[#Mesa].Bajar_MElevadora )
      Contact( #MELEV_EnMovimiento )
      I_Contact( #EstadoZona.Manual_CBx )
   END_RUNG wire#w1
   RUNG wire#powerrail
      I_Contact( #MELEV_EnMovimiento )
   END_RUNG wire#w2
   // the same network as SCL:
   #TOut_Bajar_MELEV(IN := "DB1_SalidasExterioresDeMesa".Mesa[#Mesa].Bajar_MElevadora AND #MELEV_EnMovimiento AND NOT #EstadoZona.Manual_CBx,   // "FB910_CNT_UHS"
                     R := NOT #MELEV_EnMovimiento,
                     PV := #V_TOut_MELEV,
                     BaseUnidades_ms := "CTE_BaseUnidades_1s");
END_REGION

REGION Network 54: ERROR - TimeOut Bajar Mesa Elevadora
   RUNG wire#powerrail
      Contact( #EstadoZona.Rearme_CBx )
      S_RS(operand := #EstadoVI.Err_TOut_Bajada, s1 := #TOut_Bajar_MELEV.QU)
      S_Coil( #EstadoVI.Error_Mx )
   END_RUNG
   // the same network as SCL:
   IF #EstadoZona.Rearme_CBx THEN
       #EstadoVI.Err_TOut_Bajada := FALSE;   // RS flip-flop
   END_IF;
   IF #TOut_Bajar_MELEV.QU THEN #EstadoVI.Err_TOut_Bajada := TRUE; END_IF;
   IF #EstadoVI.Err_TOut_Bajada THEN #EstadoVI.Error_Mx := TRUE; END_IF;
END_REGION

REGION Network 55: CONTROL DE TIEMPO - ERROR - Protrusión (Nota: limitacion de Valor a 1 Segundo)
   RUNG wire#powerrail
      Contact( "ON" )
      Move(in := #V_TMP_Protrusion, out1 => #V_Protrusion)
      { S7_Templates := "SrcType := Int" } GT_Contact(in1 := #V_Protrusion, in2 := 1000)
      Move(in := 1000, out1 => #V_Protrusion)
   END_RUNG
   // the same network as SCL:
   IF "ON" THEN #V_Protrusion := #V_TMP_Protrusion; END_IF;
   IF "ON" AND (#V_Protrusion > 1000) THEN #V_Protrusion := 1000; END_IF;
END_REGION

REGION Network 56: TMP - ERROR - Protrusión
   RUNG wire#powerrail
      #TMP_Protrusion(IN := wire#w6, R := wire#w7, PV := #V_Protrusion, BaseUnidades_ms := "CTE_BaseUnidades_1ms", QU =>, QD =>, CVU =>, CVD =>)
   END_RUNG
   RUNG wire#powerrail
      I_Contact( #Mx_ET10 )
      I_Contact( #Mx_ET11 )
      I_Contact( #Mx_ET12 )
      wire#w1
      I_Contact( #Mx_ET50 )
      I_Contact( #Mx_ET51 )
      wire#w2
      I_Contact( #pHsMx_PR3 )
      I_Contact( #Anular_pr3 )
   END_RUNG wire#w6
   RUNG wire#powerrail
      Contact( #Selec_M1M2_Entrada )
   END_RUNG wire#w1
   RUNG wire#w1
      Contact( #Selec_M1M2_Salida )
   END_RUNG wire#w2
   RUNG wire#powerrail
      I_Contact( #MELEV_UP )
      I_Contact( #MELEV_DW )
   END_RUNG wire#w2
   RUNG wire#powerrail
      I_Contact( #Mx_ET10 )
      I_Contact( #Mx_ET11 )
      I_Contact( #Mx_ET12 )
      wire#w3
      I_Contact( #Mx_ET50 )
      I_Contact( #Mx_ET51 )
      wire#w4
      I_Contact( #pHsMx_PR1 )
      I_Contact( #Anular_pr1 )
   END_RUNG wire#w6
   RUNG wire#powerrail
      Contact( #Selec_M3M4_Entrada )
   END_RUNG wire#w3
   RUNG wire#w3
      Contact( #Selec_M3M4_Salida )
   END_RUNG wire#w4
   RUNG wire#powerrail
      I_Contact( #MELEV_UP )
      I_Contact( #MELEV_DW )
   END_RUNG wire#w4
   RUNG wire#powerrail
      I_Contact( #pHsMx_PR1 )
      I_Contact( #Anular_pr1 )
      wire#w5
      Contact( #EstadoZona.Manual_CBx )
   END_RUNG wire#w6
   RUNG wire#powerrail
      I_Contact( #pHsMx_PR3 )
      I_Contact( #Anular_pr3 )
   END_RUNG wire#w5
   RUNG wire#powerrail
      Contact( #pHsMx_PR1 )
      Contact( #pHsMx_PR3 )
   END_RUNG wire#w7
   // the same network as SCL:
   #TMP_Protrusion(IN := (((((NOT #Mx_ET10 AND NOT #Mx_ET11 AND NOT #Mx_ET12) OR #Selec_M1M2_Entrada) AND ((NOT #Mx_ET50 AND NOT #Mx_ET51) OR #Selec_M1M2_Salida)) OR (NOT #MELEV_UP AND NOT #MELEV_DW)) AND NOT #pHsMx_PR3 AND NOT #Anular_pr3) OR (((((NOT #Mx_ET10 AND NOT #Mx_ET11 AND NOT #Mx_ET12) OR #Selec_M3M4_Entrada) AND ((NOT #Mx_ET50 AND NOT #Mx_ET51) OR #Selec_M3M4_Salida)) OR (NOT #MELEV_UP AND NOT #MELEV_DW)) AND NOT #pHsMx_PR1 AND NOT #Anular_pr1) OR (((NOT #pHsMx_PR1 AND NOT #Anular_pr1) OR (NOT #pHsMx_PR3 AND NOT #Anular_pr3)) AND #EstadoZona.Manual_CBx),   // "FB910_CNT_UHS"
                   R := #pHsMx_PR1 AND #pHsMx_PR3,
                   PV := #V_Protrusion,
                   BaseUnidades_ms := "CTE_BaseUnidades_1ms");
END_REGION

REGION Network 57: ERROR - Protrusión
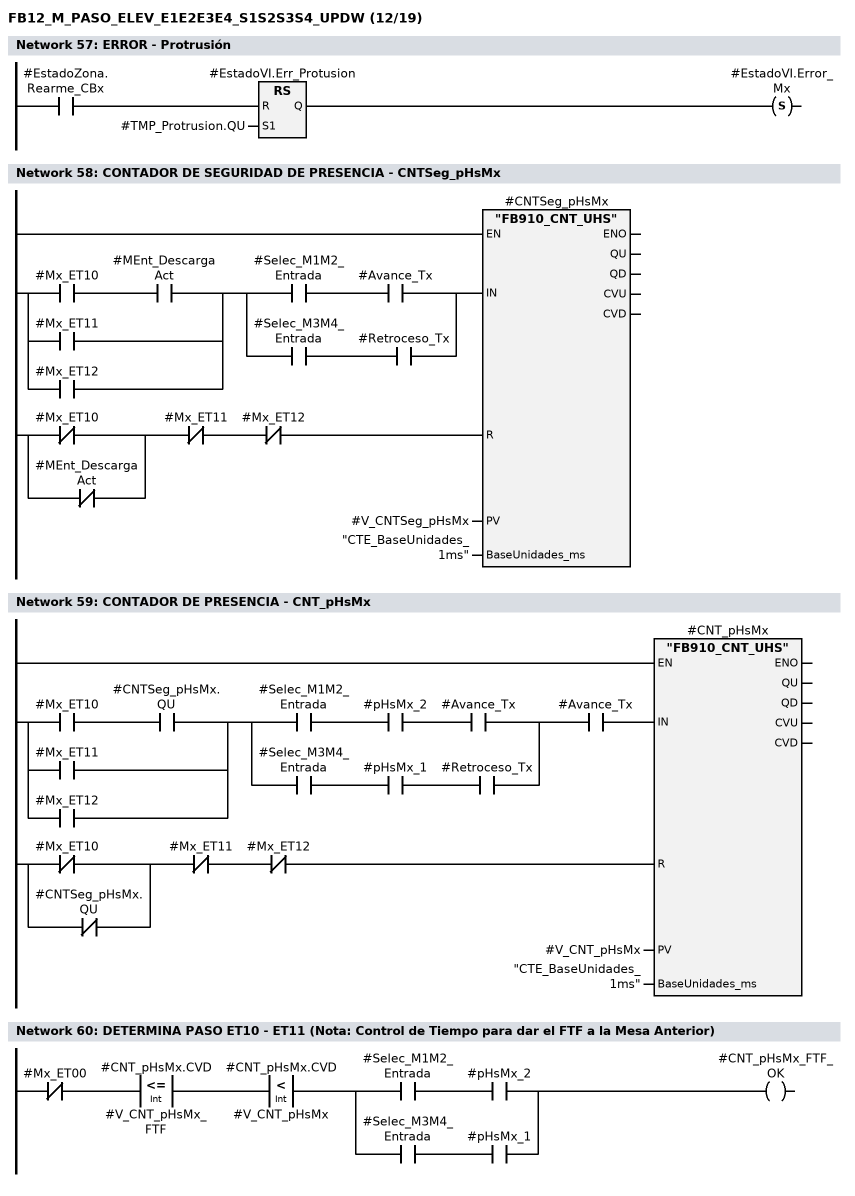
   RUNG wire#powerrail
      Contact( #EstadoZona.Rearme_CBx )
      S_RS(operand := #EstadoVI.Err_Protusion, s1 := #TMP_Protrusion.QU)
      S_Coil( #EstadoVI.Error_Mx )
   END_RUNG
   // the same network as SCL:
   IF #EstadoZona.Rearme_CBx THEN
       #EstadoVI.Err_Protusion := FALSE;   // RS flip-flop
   END_IF;
   IF #TMP_Protrusion.QU THEN #EstadoVI.Err_Protusion := TRUE; END_IF;
   IF #EstadoVI.Err_Protusion THEN #EstadoVI.Error_Mx := TRUE; END_IF;
END_REGION

REGION Network 58: CONTADOR DE SEGURIDAD DE PRESENCIA - CNTSeg_pHsMx
   RUNG wire#powerrail
      #CNTSeg_pHsMx(IN := wire#w2, R := wire#w4, PV := #V_CNTSeg_pHsMx, BaseUnidades_ms := "CTE_BaseUnidades_1ms", QU =>, QD =>, CVU =>, CVD =>)
   END_RUNG
   RUNG wire#powerrail
      Contact( #Mx_ET10 )
      Contact( #MEnt_DescargaAct )
      wire#w1
      Contact( #Selec_M1M2_Entrada )
      Contact( #Avance_Tx )
   END_RUNG wire#w2
   RUNG wire#powerrail
      Contact( #Mx_ET11 )
   END_RUNG wire#w1
   RUNG wire#powerrail
      Contact( #Mx_ET12 )
   END_RUNG wire#w1
   RUNG wire#w1
      Contact( #Selec_M3M4_Entrada )
      Contact( #Retroceso_Tx )
   END_RUNG wire#w2
   RUNG wire#powerrail
      I_Contact( #Mx_ET10 )
      wire#w3
      I_Contact( #Mx_ET11 )
      I_Contact( #Mx_ET12 )
   END_RUNG wire#w4
   RUNG wire#powerrail
      I_Contact( #MEnt_DescargaAct )
   END_RUNG wire#w3
   // the same network as SCL:
   #CNTSeg_pHsMx(IN := ((#Mx_ET10 AND #MEnt_DescargaAct) OR #Mx_ET11 OR #Mx_ET12) AND ((#Selec_M1M2_Entrada AND #Avance_Tx) OR (#Selec_M3M4_Entrada AND #Retroceso_Tx)),   // "FB910_CNT_UHS"
                 R := (NOT #Mx_ET10 OR NOT #MEnt_DescargaAct) AND NOT #Mx_ET11 AND NOT #Mx_ET12,
                 PV := #V_CNTSeg_pHsMx,
                 BaseUnidades_ms := "CTE_BaseUnidades_1ms");
END_REGION

REGION Network 59: CONTADOR DE PRESENCIA - CNT_pHsMx
   RUNG wire#powerrail
      #CNT_pHsMx(IN := wire#w3, R := wire#w5, PV := #V_CNT_pHsMx, BaseUnidades_ms := "CTE_BaseUnidades_1ms", QU =>, QD =>, CVU =>, CVD =>)
   END_RUNG
   RUNG wire#powerrail
      Contact( #Mx_ET10 )
      Contact( #CNTSeg_pHsMx.QU )
      wire#w1
      Contact( #Selec_M1M2_Entrada )
      Contact( #pHsMx_2 )
      Contact( #Avance_Tx )
      wire#w2
      Contact( #Avance_Tx )
   END_RUNG wire#w3
   RUNG wire#powerrail
      Contact( #Mx_ET11 )
   END_RUNG wire#w1
   RUNG wire#powerrail
      Contact( #Mx_ET12 )
   END_RUNG wire#w1
   RUNG wire#w1
      Contact( #Selec_M3M4_Entrada )
      Contact( #pHsMx_1 )
      Contact( #Retroceso_Tx )
   END_RUNG wire#w2
   RUNG wire#powerrail
      I_Contact( #Mx_ET10 )
      wire#w4
      I_Contact( #Mx_ET11 )
      I_Contact( #Mx_ET12 )
   END_RUNG wire#w5
   RUNG wire#powerrail
      I_Contact( #CNTSeg_pHsMx.QU )
   END_RUNG wire#w4
   // the same network as SCL:
   #CNT_pHsMx(IN := ((#Mx_ET10 AND #CNTSeg_pHsMx.QU) OR #Mx_ET11 OR #Mx_ET12) AND ((#Selec_M1M2_Entrada AND #pHsMx_2 AND #Avance_Tx) OR (#Selec_M3M4_Entrada AND #pHsMx_1 AND #Retroceso_Tx)) AND #Avance_Tx,   // "FB910_CNT_UHS"
              R := (NOT #Mx_ET10 OR NOT #CNTSeg_pHsMx.QU) AND NOT #Mx_ET11 AND NOT #Mx_ET12,
              PV := #V_CNT_pHsMx,
              BaseUnidades_ms := "CTE_BaseUnidades_1ms");
END_REGION

REGION Network 60: DETERMINA PASO ET10 - ET11 (Nota: Control de Tiempo para dar el FTF a la Mesa Anterior)
   RUNG wire#powerrail
      I_Contact( #Mx_ET00 )
      { S7_Templates := "SrcType := Int" } LE_Contact(in1 := #CNT_pHsMx.CVD, in2 := #V_CNT_pHsMx_FTF)
      { S7_Templates := "SrcType := Int" } LT_Contact(in1 := #CNT_pHsMx.CVD, in2 := #V_CNT_pHsMx)
      wire#w1
      Contact( #Selec_M1M2_Entrada )
      Contact( #pHsMx_2 )
      wire#w2
      Coil( #CNT_pHsMx_FTF_OK )
   END_RUNG
   RUNG wire#w1
      Contact( #Selec_M3M4_Entrada )
      Contact( #pHsMx_1 )
   END_RUNG wire#w2
   // the same network as SCL:
   #CNT_pHsMx_FTF_OK := NOT #Mx_ET00 AND (#CNT_pHsMx.CVD <= #V_CNT_pHsMx_FTF) AND (#CNT_pHsMx.CVD < #V_CNT_pHsMx) AND ((#Selec_M1M2_Entrada AND #pHsMx_2) OR (#Selec_M3M4_Entrada AND #pHsMx_1));
END_REGION

REGION Network 61: CONTADOR SEGURIDAD DE AUSENCIA - CNTSeg_ApHsMx ??????? RESTAR VALOR DE POSICIONAMIENTO
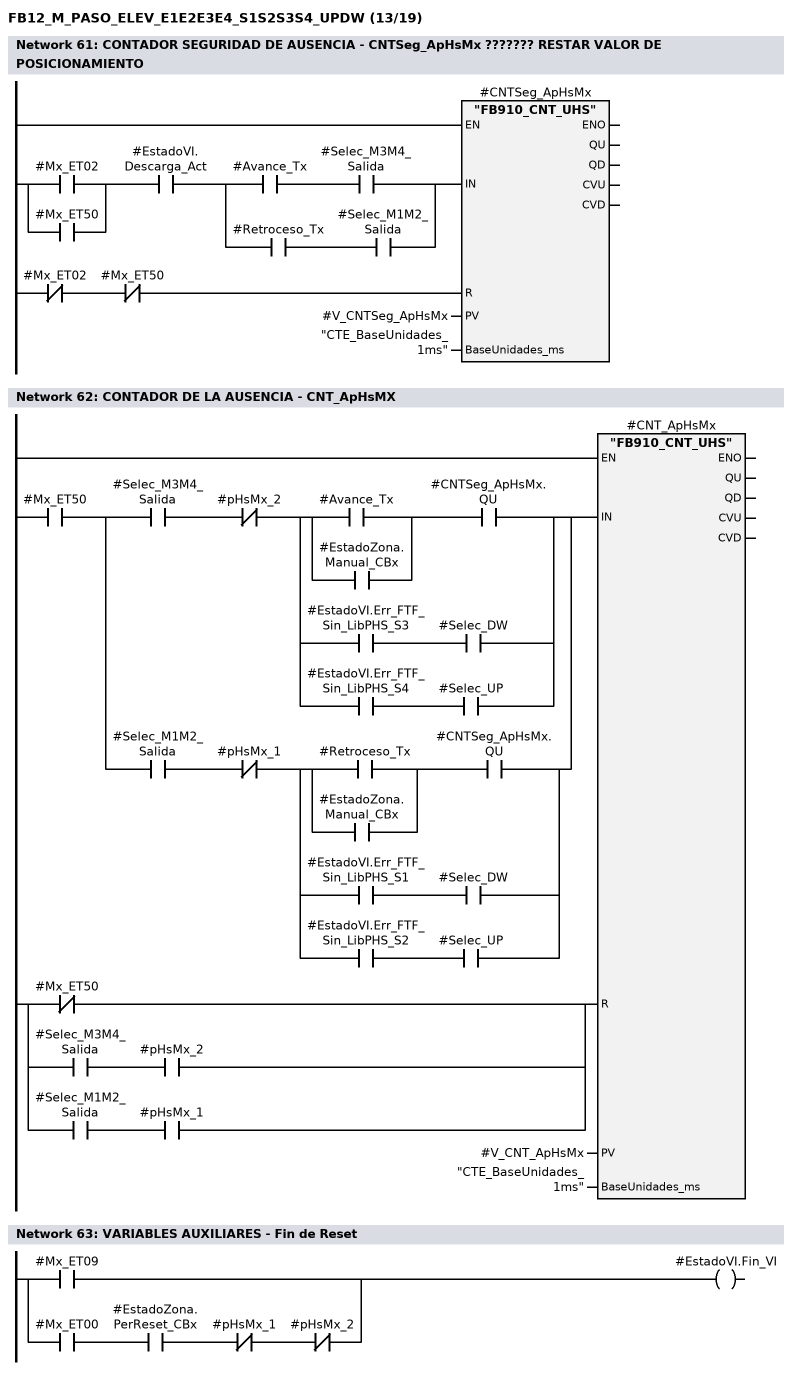
   RUNG wire#powerrail
      #CNTSeg_ApHsMx(IN := wire#w3, R := wire#w4, PV := #V_CNTSeg_ApHsMx, BaseUnidades_ms := "CTE_BaseUnidades_1ms", QU =>, QD =>, CVU =>, CVD =>)
   END_RUNG
   RUNG wire#powerrail
      Contact( #Mx_ET02 )
      wire#w1
      Contact( #EstadoVI.Descarga_Act )
      wire#w2
      Contact( #Avance_Tx )
      Contact( #Selec_M3M4_Salida )
   END_RUNG wire#w3
   RUNG wire#powerrail
      Contact( #Mx_ET50 )
   END_RUNG wire#w1
   RUNG wire#w2
      Contact( #Retroceso_Tx )
      Contact( #Selec_M1M2_Salida )
   END_RUNG wire#w3
   RUNG wire#powerrail
      I_Contact( #Mx_ET02 )
      I_Contact( #Mx_ET50 )
   END_RUNG wire#w4
   // the same network as SCL:
   #CNTSeg_ApHsMx(IN := (#Mx_ET02 OR #Mx_ET50) AND #EstadoVI.Descarga_Act AND ((#Avance_Tx AND #Selec_M3M4_Salida) OR (#Retroceso_Tx AND #Selec_M1M2_Salida)),   // "FB910_CNT_UHS"
                  R := NOT #Mx_ET02 AND NOT #Mx_ET50,
                  PV := #V_CNTSeg_ApHsMx,
                  BaseUnidades_ms := "CTE_BaseUnidades_1ms");
END_REGION

REGION Network 62: CONTADOR DE LA AUSENCIA - CNT_ApHsMX
   RUNG wire#powerrail
      #CNT_ApHsMx(IN := wire#w6, R := wire#w7, PV := #V_CNT_ApHsMx, BaseUnidades_ms := "CTE_BaseUnidades_1ms", QU =>, QD =>, CVU =>, CVD =>)
   END_RUNG
   RUNG wire#powerrail
      Contact( #Mx_ET50 )
      wire#w1
      Contact( #Selec_M3M4_Salida )
      I_Contact( #pHsMx_2 )
      wire#w2
      Contact( #Avance_Tx )
      wire#w3
      Contact( #CNTSeg_ApHsMx.QU )
   END_RUNG wire#w6
   RUNG wire#w2
      Contact( #EstadoZona.Manual_CBx )
   END_RUNG wire#w3
   RUNG wire#w2
      Contact( #EstadoVI.Err_FTF_Sin_LibPHS_S3 )
      Contact( #Selec_DW )
   END_RUNG wire#w6
   RUNG wire#w2
      Contact( #EstadoVI.Err_FTF_Sin_LibPHS_S4 )
      Contact( #Selec_UP )
   END_RUNG wire#w6
   RUNG wire#w1
      Contact( #Selec_M1M2_Salida )
      I_Contact( #pHsMx_1 )
      wire#w4
      Contact( #Retroceso_Tx )
      wire#w5
      Contact( #CNTSeg_ApHsMx.QU )
   END_RUNG wire#w6
   RUNG wire#w4
      Contact( #EstadoZona.Manual_CBx )
   END_RUNG wire#w5
   RUNG wire#w4
      Contact( #EstadoVI.Err_FTF_Sin_LibPHS_S1 )
      Contact( #Selec_DW )
   END_RUNG wire#w6
   RUNG wire#w4
      Contact( #EstadoVI.Err_FTF_Sin_LibPHS_S2 )
      Contact( #Selec_UP )
   END_RUNG wire#w6
   RUNG wire#powerrail
      I_Contact( #Mx_ET50 )
   END_RUNG wire#w7
   RUNG wire#powerrail
      Contact( #Selec_M3M4_Salida )
      Contact( #pHsMx_2 )
   END_RUNG wire#w7
   RUNG wire#powerrail
      Contact( #Selec_M1M2_Salida )
      Contact( #pHsMx_1 )
   END_RUNG wire#w7
   // the same network as SCL:
   #CNT_ApHsMx(IN := #Mx_ET50 AND ((#Selec_M3M4_Salida AND NOT #pHsMx_2 AND (((#Avance_Tx OR #EstadoZona.Manual_CBx) AND #CNTSeg_ApHsMx.QU) OR (#EstadoVI.Err_FTF_Sin_LibPHS_S3 AND #Selec_DW) OR (#EstadoVI.Err_FTF_Sin_LibPHS_S4 AND #Selec_UP))) OR (#Selec_M1M2_Salida AND NOT #pHsMx_1 AND (((#Retroceso_Tx OR #EstadoZona.Manual_CBx) AND #CNTSeg_ApHsMx.QU) OR (#EstadoVI.Err_FTF_Sin_LibPHS_S1 AND #Selec_DW) OR (#EstadoVI.Err_FTF_Sin_LibPHS_S2 AND #Selec_UP)))),   // "FB910_CNT_UHS"
               R := NOT #Mx_ET50 OR (#Selec_M3M4_Salida AND #pHsMx_2) OR (#Selec_M1M2_Salida AND #pHsMx_1),
               PV := #V_CNT_ApHsMx,
               BaseUnidades_ms := "CTE_BaseUnidades_1ms");
END_REGION

REGION Network 63: VARIABLES AUXILIARES - Fin de Reset
   RUNG wire#powerrail
      Contact( #Mx_ET09 )
      wire#w1
      Coil( #EstadoVI.Fin_VI )
   END_RUNG
   RUNG wire#powerrail
      Contact( #Mx_ET00 )
      Contact( #EstadoZona.PerReset_CBx )
      I_Contact( #pHsMx_1 )
      I_Contact( #pHsMx_2 )
   END_RUNG wire#w1
   // the same network as SCL:
   #EstadoVI.Fin_VI := #Mx_ET09 OR (#Mx_ET00 AND #EstadoZona.PerReset_CBx AND NOT #pHsMx_1 AND NOT #pHsMx_2);
END_REGION

REGION Network 64: VARIABLES AUXILIARES - Fin de Paro blando
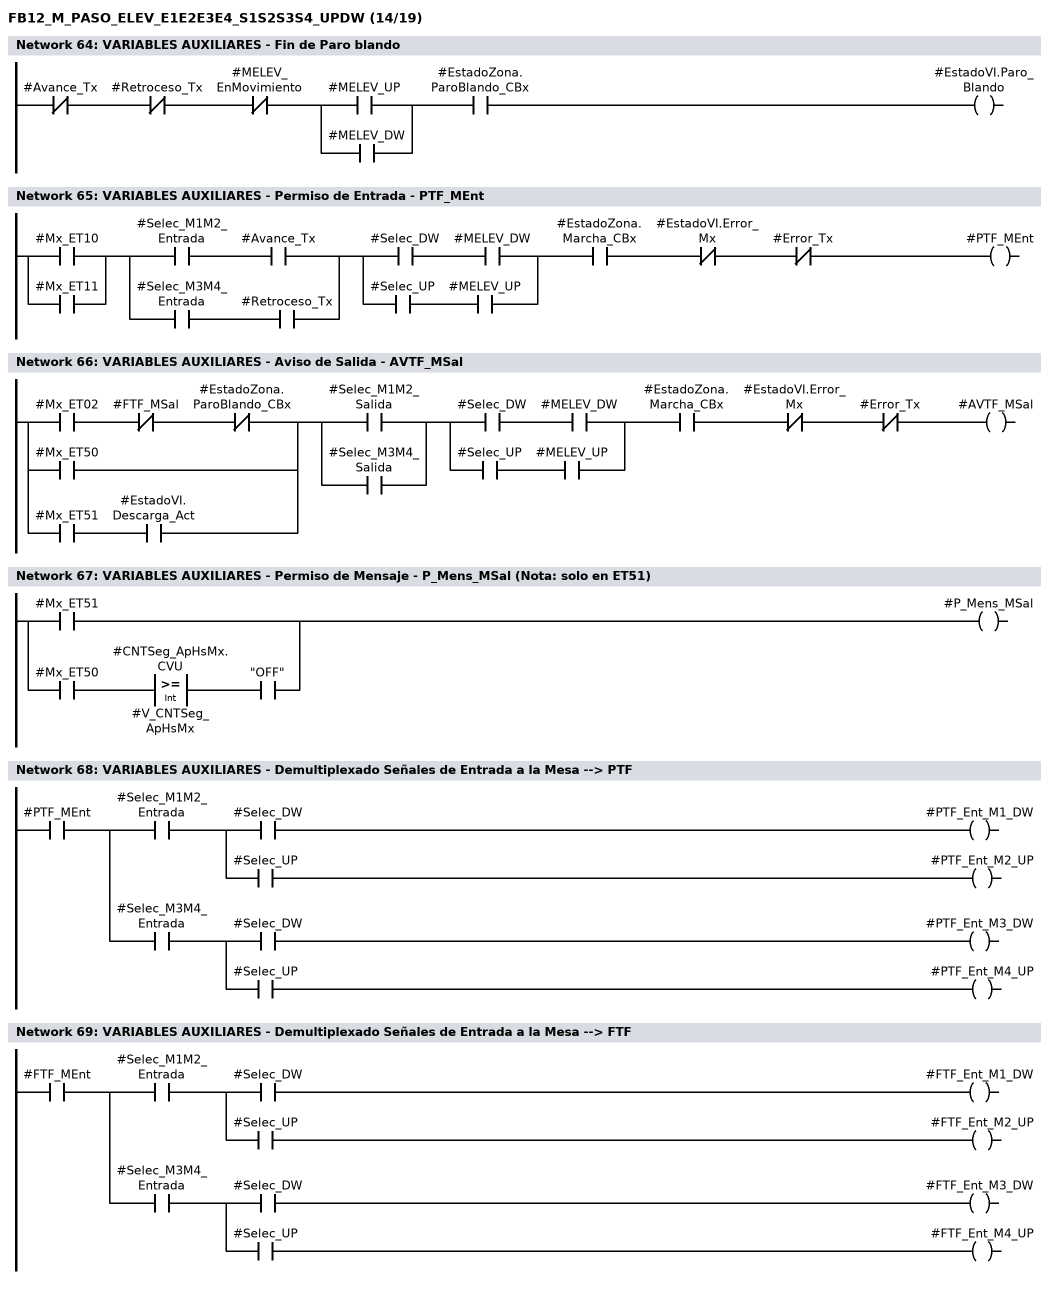
   RUNG wire#powerrail
      I_Contact( #Avance_Tx )
      I_Contact( #Retroceso_Tx )
      I_Contact( #MELEV_EnMovimiento )
      wire#w1
      Contact( #MELEV_UP )
      wire#w2
      Contact( #EstadoZona.ParoBlando_CBx )
      Coil( #EstadoVI.Paro_Blando )
   END_RUNG
   RUNG wire#w1
      Contact( #MELEV_DW )
   END_RUNG wire#w2
   // the same network as SCL:
   #EstadoVI.Paro_Blando := NOT #Avance_Tx AND NOT #Retroceso_Tx AND NOT #MELEV_EnMovimiento AND (#MELEV_UP OR #MELEV_DW) AND #EstadoZona.ParoBlando_CBx;
END_REGION

REGION Network 65: VARIABLES AUXILIARES - Permiso de Entrada - PTF_MEnt
   RUNG wire#powerrail
      Contact( #Mx_ET10 )
      wire#w1
      Contact( #Selec_M1M2_Entrada )
      Contact( #Avance_Tx )
      wire#w2
      Contact( #Selec_DW )
      Contact( #MELEV_DW )
      wire#w3
      Contact( #EstadoZona.Marcha_CBx )
      I_Contact( #EstadoVI.Error_Mx )
      I_Contact( #Error_Tx )
      Coil( #PTF_MEnt )
   END_RUNG
   RUNG wire#powerrail
      Contact( #Mx_ET11 )
   END_RUNG wire#w1
   RUNG wire#w1
      Contact( #Selec_M3M4_Entrada )
      Contact( #Retroceso_Tx )
   END_RUNG wire#w2
   RUNG wire#w2
      Contact( #Selec_UP )
      Contact( #MELEV_UP )
   END_RUNG wire#w3
   // the same network as SCL:
   #PTF_MEnt := (#Mx_ET10 OR #Mx_ET11) AND ((#Selec_M1M2_Entrada AND #Avance_Tx) OR (#Selec_M3M4_Entrada AND #Retroceso_Tx)) AND ((#Selec_DW AND #MELEV_DW) OR (#Selec_UP AND #MELEV_UP)) AND #EstadoZona.Marcha_CBx AND NOT #EstadoVI.Error_Mx AND NOT #Error_Tx;
END_REGION

REGION Network 66: VARIABLES AUXILIARES - Aviso de Salida - AVTF_MSal
   RUNG wire#powerrail
      Contact( #Mx_ET02 )
      I_Contact( #FTF_MSal )
      I_Contact( #EstadoZona.ParoBlando_CBx )
      wire#w1
      Contact( #Selec_M1M2_Salida )
      wire#w2
      Contact( #Selec_DW )
      Contact( #MELEV_DW )
      wire#w3
      Contact( #EstadoZona.Marcha_CBx )
      I_Contact( #EstadoVI.Error_Mx )
      I_Contact( #Error_Tx )
      Coil( #AVTF_MSal )
   END_RUNG
   RUNG wire#powerrail
      Contact( #Mx_ET50 )
   END_RUNG wire#w1
   RUNG wire#powerrail
      Contact( #Mx_ET51 )
      Contact( #EstadoVI.Descarga_Act )
   END_RUNG wire#w1
   RUNG wire#w1
      Contact( #Selec_M3M4_Salida )
   END_RUNG wire#w2
   RUNG wire#w2
      Contact( #Selec_UP )
      Contact( #MELEV_UP )
   END_RUNG wire#w3
   // the same network as SCL:
   #AVTF_MSal := ((#Mx_ET02 AND NOT #FTF_MSal AND NOT #EstadoZona.ParoBlando_CBx) OR #Mx_ET50 OR (#Mx_ET51 AND #EstadoVI.Descarga_Act)) AND (#Selec_M1M2_Salida OR #Selec_M3M4_Salida) AND ((#Selec_DW AND #MELEV_DW) OR (#Selec_UP AND #MELEV_UP)) AND #EstadoZona.Marcha_CBx AND NOT #EstadoVI.Error_Mx AND NOT #Error_Tx;
END_REGION

REGION Network 67: VARIABLES AUXILIARES - Permiso de Mensaje - P_Mens_MSal (Nota: solo en ET51)
   RUNG wire#powerrail
      Contact( #Mx_ET51 )
      wire#w1
      Coil( #P_Mens_MSal )
   END_RUNG
   RUNG wire#powerrail
      Contact( #Mx_ET50 )
      { S7_Templates := "SrcType := Int" } GE_Contact(in1 := #CNTSeg_ApHsMx.CVU, in2 := #V_CNTSeg_ApHsMx)
      Contact( "OFF" )
   END_RUNG wire#w1
   // the same network as SCL:
   #P_Mens_MSal := #Mx_ET51 OR (#Mx_ET50 AND (#CNTSeg_ApHsMx.CVU >= #V_CNTSeg_ApHsMx) AND "OFF");
END_REGION

REGION Network 68: VARIABLES AUXILIARES - Demultiplexado Señales de Entrada a la Mesa --> PTF
   RUNG wire#powerrail
      Contact( #PTF_MEnt )
      wire#w1
      Contact( #Selec_M1M2_Entrada )
      wire#w2
      Contact( #Selec_DW )
      Coil( #PTF_Ent_M1_DW )
   END_RUNG
   RUNG wire#w2
      Contact( #Selec_UP )
      Coil( #PTF_Ent_M2_UP )
   END_RUNG
   RUNG wire#w1
      Contact( #Selec_M3M4_Entrada )
      wire#w3
      Contact( #Selec_DW )
      Coil( #PTF_Ent_M3_DW )
   END_RUNG
   RUNG wire#w3
      Contact( #Selec_UP )
      Coil( #PTF_Ent_M4_UP )
   END_RUNG
   // the same network as SCL:
   #_w1 := #PTF_MEnt AND #Selec_M1M2_Entrada;
   #PTF_Ent_M1_DW := #_w1 AND #Selec_DW;
   #PTF_Ent_M2_UP := #_w1 AND #Selec_UP;
   #_w2 := #PTF_MEnt AND #Selec_M3M4_Entrada;
   #PTF_Ent_M3_DW := #_w2 AND #Selec_DW;
   #PTF_Ent_M4_UP := #_w2 AND #Selec_UP;
END_REGION

REGION Network 69: VARIABLES AUXILIARES - Demultiplexado Señales de Entrada a la Mesa --> FTF
   RUNG wire#powerrail
      Contact( #FTF_MEnt )
      wire#w1
      Contact( #Selec_M1M2_Entrada )
      wire#w2
      Contact( #Selec_DW )
      Coil( #FTF_Ent_M1_DW )
   END_RUNG
   RUNG wire#w2
      Contact( #Selec_UP )
      Coil( #FTF_Ent_M2_UP )
   END_RUNG
   RUNG wire#w1
      Contact( #Selec_M3M4_Entrada )
      wire#w3
      Contact( #Selec_DW )
      Coil( #FTF_Ent_M3_DW )
   END_RUNG
   RUNG wire#w3
      Contact( #Selec_UP )
      Coil( #FTF_Ent_M4_UP )
   END_RUNG
   // the same network as SCL:
   #_w1 := #FTF_MEnt AND #Selec_M1M2_Entrada;
   #FTF_Ent_M1_DW := #_w1 AND #Selec_DW;
   #FTF_Ent_M2_UP := #_w1 AND #Selec_UP;
   #_w2 := #FTF_MEnt AND #Selec_M3M4_Entrada;
   #FTF_Ent_M3_DW := #_w2 AND #Selec_DW;
   #FTF_Ent_M4_UP := #_w2 AND #Selec_UP;
END_REGION

REGION Network 70: VARIABLES AUXILIARES - Demultiplexado Señales de Salida de la Mesa --> ATF
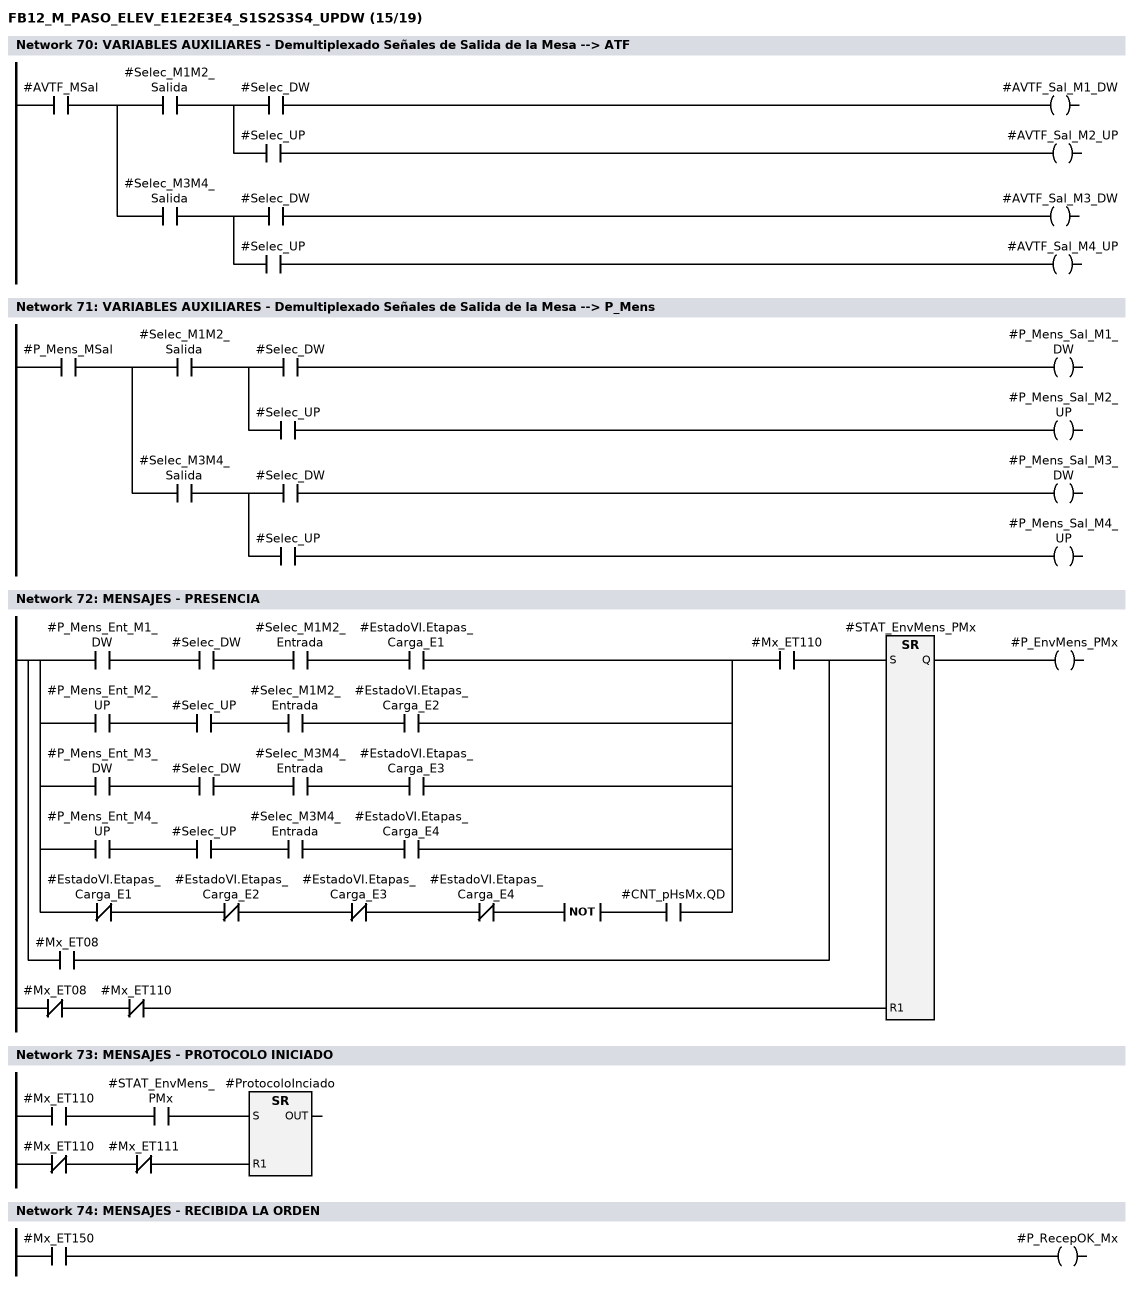
   RUNG wire#powerrail
      Contact( #AVTF_MSal )
      wire#w1
      Contact( #Selec_M1M2_Salida )
      wire#w2
      Contact( #Selec_DW )
      Coil( #AVTF_Sal_M1_DW )
   END_RUNG
   RUNG wire#w2
      Contact( #Selec_UP )
      Coil( #AVTF_Sal_M2_UP )
   END_RUNG
   RUNG wire#w1
      Contact( #Selec_M3M4_Salida )
      wire#w3
      Contact( #Selec_DW )
      Coil( #AVTF_Sal_M3_DW )
   END_RUNG
   RUNG wire#w3
      Contact( #Selec_UP )
      Coil( #AVTF_Sal_M4_UP )
   END_RUNG
   // the same network as SCL:
   #_w1 := #AVTF_MSal AND #Selec_M1M2_Salida;
   #AVTF_Sal_M1_DW := #_w1 AND #Selec_DW;
   #AVTF_Sal_M2_UP := #_w1 AND #Selec_UP;
   #_w2 := #AVTF_MSal AND #Selec_M3M4_Salida;
   #AVTF_Sal_M3_DW := #_w2 AND #Selec_DW;
   #AVTF_Sal_M4_UP := #_w2 AND #Selec_UP;
END_REGION

REGION Network 71: VARIABLES AUXILIARES - Demultiplexado Señales de Salida de la Mesa --> P_Mens
   RUNG wire#powerrail
      Contact( #P_Mens_MSal )
      wire#w1
      Contact( #Selec_M1M2_Salida )
      wire#w2
      Contact( #Selec_DW )
      Coil( #P_Mens_Sal_M1_DW )
   END_RUNG
   RUNG wire#w2
      Contact( #Selec_UP )
      Coil( #P_Mens_Sal_M2_UP )
   END_RUNG
   RUNG wire#w1
      Contact( #Selec_M3M4_Salida )
      wire#w3
      Contact( #Selec_DW )
      Coil( #P_Mens_Sal_M3_DW )
   END_RUNG
   RUNG wire#w3
      Contact( #Selec_UP )
      Coil( #P_Mens_Sal_M4_UP )
   END_RUNG
   // the same network as SCL:
   #_w1 := #P_Mens_MSal AND #Selec_M1M2_Salida;
   #P_Mens_Sal_M1_DW := #_w1 AND #Selec_DW;
   #P_Mens_Sal_M2_UP := #_w1 AND #Selec_UP;
   #_w2 := #P_Mens_MSal AND #Selec_M3M4_Salida;
   #P_Mens_Sal_M3_DW := #_w2 AND #Selec_DW;
   #P_Mens_Sal_M4_UP := #_w2 AND #Selec_UP;
END_REGION

REGION Network 72: MENSAJES - PRESENCIA
   RUNG wire#powerrail
      Contact( #P_Mens_Ent_M1_DW )
      Contact( #Selec_DW )
      Contact( #Selec_M1M2_Entrada )
      Contact( #EstadoVI.Etapas_Carga_E1 )
      wire#w1
      Contact( #Mx_ET110 )
      wire#w2
      S_SR(operand := #STAT_EnvMens_PMx, r1 := wire#w3)
      Coil( #P_EnvMens_PMx )
   END_RUNG
   RUNG wire#powerrail
      Contact( #P_Mens_Ent_M2_UP )
      Contact( #Selec_UP )
      Contact( #Selec_M1M2_Entrada )
      Contact( #EstadoVI.Etapas_Carga_E2 )
   END_RUNG wire#w1
   RUNG wire#powerrail
      Contact( #P_Mens_Ent_M3_DW )
      Contact( #Selec_DW )
      Contact( #Selec_M3M4_Entrada )
      Contact( #EstadoVI.Etapas_Carga_E3 )
   END_RUNG wire#w1
   RUNG wire#powerrail
      Contact( #P_Mens_Ent_M4_UP )
      Contact( #Selec_UP )
      Contact( #Selec_M3M4_Entrada )
      Contact( #EstadoVI.Etapas_Carga_E4 )
   END_RUNG wire#w1
   RUNG wire#powerrail
      I_Contact( #EstadoVI.Etapas_Carga_E1 )
      I_Contact( #EstadoVI.Etapas_Carga_E2 )
      I_Contact( #EstadoVI.Etapas_Carga_E3 )
      I_Contact( #EstadoVI.Etapas_Carga_E4 )
      Not()
      Contact( #CNT_pHsMx.QD )
   END_RUNG wire#w1
   RUNG wire#powerrail
      Contact( #Mx_ET08 )
   END_RUNG wire#w2
   RUNG wire#powerrail
      I_Contact( #Mx_ET08 )
      I_Contact( #Mx_ET110 )
   END_RUNG wire#w3
   // the same network as SCL:
   IF (((#P_Mens_Ent_M1_DW AND #Selec_DW AND #Selec_M1M2_Entrada AND #EstadoVI.Etapas_Carga_E1) OR (#P_Mens_Ent_M2_UP AND #Selec_UP AND #Selec_M1M2_Entrada AND #EstadoVI.Etapas_Carga_E2) OR (#P_Mens_Ent_M3_DW AND #Selec_DW AND #Selec_M3M4_Entrada AND #EstadoVI.Etapas_Carga_E3) OR (#P_Mens_Ent_M4_UP AND #Selec_UP AND #Selec_M3M4_Entrada AND #EstadoVI.Etapas_Carga_E4) OR (NOT (NOT #EstadoVI.Etapas_Carga_E1 AND NOT #EstadoVI.Etapas_Carga_E2 AND NOT #EstadoVI.Etapas_Carga_E3 AND NOT #EstadoVI.Etapas_Carga_E4) AND #CNT_pHsMx.QD)) AND #Mx_ET110) OR #Mx_ET08 THEN
       #STAT_EnvMens_PMx := TRUE;   // SR flip-flop
   END_IF;
   IF NOT #Mx_ET08 AND NOT #Mx_ET110 THEN #STAT_EnvMens_PMx := FALSE; END_IF;
   #P_EnvMens_PMx := #STAT_EnvMens_PMx;
END_REGION

REGION Network 73: MENSAJES - PROTOCOLO INICIADO
   RUNG wire#powerrail
      Contact( #Mx_ET110 )
      Contact( #STAT_EnvMens_PMx )
      S_SR(operand := #ProtocoloInciado, r1 := wire#w1)
   END_RUNG
   RUNG wire#powerrail
      I_Contact( #Mx_ET110 )
      I_Contact( #Mx_ET111 )
   END_RUNG wire#w1
   // the same network as SCL:
   IF #Mx_ET110 AND #STAT_EnvMens_PMx THEN
       #ProtocoloInciado := TRUE;   // SR flip-flop
   END_IF;
   IF NOT #Mx_ET110 AND NOT #Mx_ET111 THEN #ProtocoloInciado := FALSE; END_IF;
END_REGION

REGION Network 74: MENSAJES - RECIBIDA LA ORDEN
   RUNG wire#powerrail
      Contact( #Mx_ET150 )
      Coil( #P_RecepOK_Mx )
   END_RUNG
   // the same network as SCL:
   #P_RecepOK_Mx := #Mx_ET150;
END_REGION

REGION Network 75: SALIDAS - Avanzar E1E3
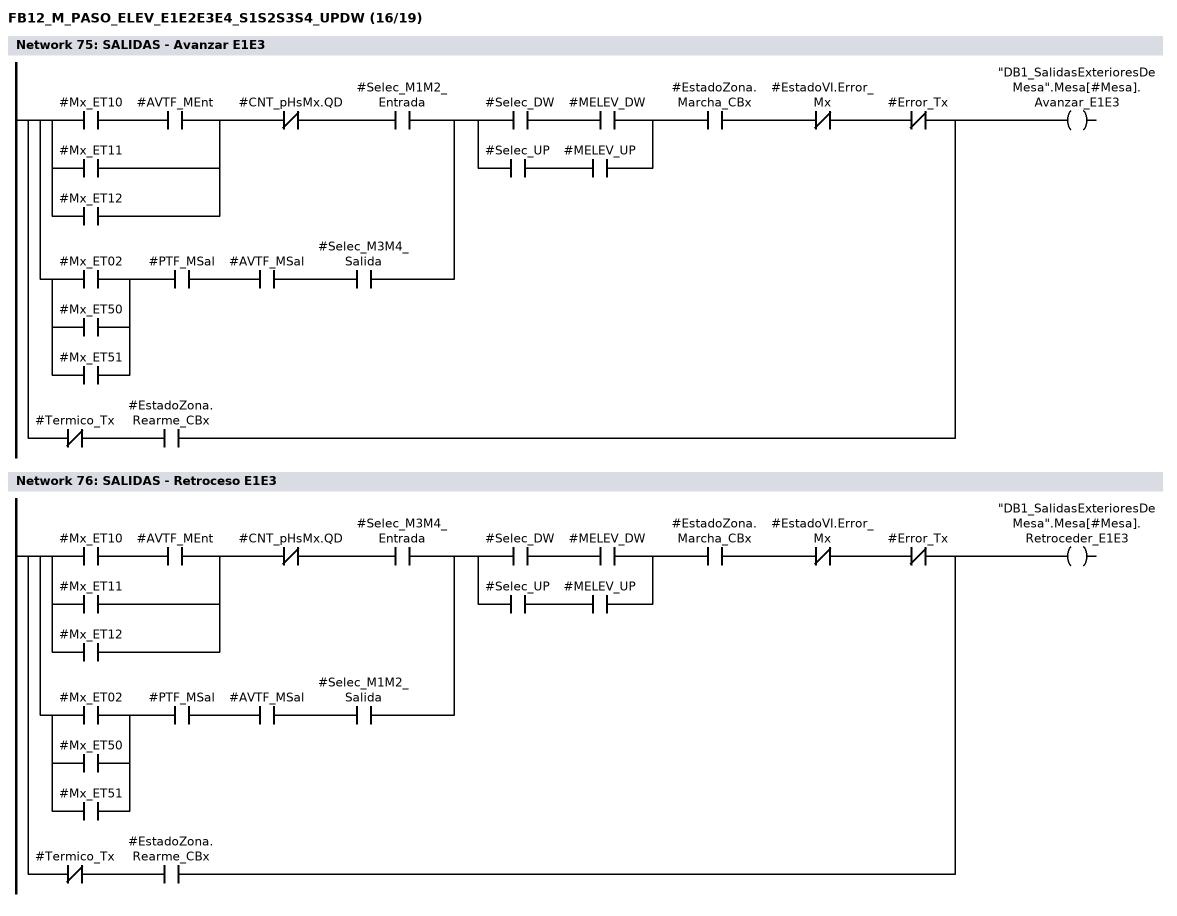
   RUNG wire#powerrail
      Contact( #Mx_ET10 )
      Contact( #AVTF_MEnt )
      wire#w1
      I_Contact( #CNT_pHsMx.QD )
      Contact( #Selec_M1M2_Entrada )
      wire#w2
      Contact( #Selec_DW )
      Contact( #MELEV_DW )
      wire#w4
      Contact( #EstadoZona.Marcha_CBx )
      I_Contact( #EstadoVI.Error_Mx )
      I_Contact( #Error_Tx )
      wire#w5
      Coil( "DB1_SalidasExterioresDeMesa".Mesa[#Mesa].Avanzar_E1E3 )
   END_RUNG
   RUNG wire#powerrail
      Contact( #Mx_ET11 )
   END_RUNG wire#w1
   RUNG wire#powerrail
      Contact( #Mx_ET12 )
   END_RUNG wire#w1
   RUNG wire#powerrail
      Contact( #Mx_ET02 )
      wire#w3
      Contact( #PTF_MSal )
      Contact( #AVTF_MSal )
      Contact( #Selec_M3M4_Salida )
   END_RUNG wire#w2
   RUNG wire#powerrail
      Contact( #Mx_ET50 )
   END_RUNG wire#w3
   RUNG wire#powerrail
      Contact( #Mx_ET51 )
   END_RUNG wire#w3
   RUNG wire#w2
      Contact( #Selec_UP )
      Contact( #MELEV_UP )
   END_RUNG wire#w4
   RUNG wire#powerrail
      I_Contact( #Termico_Tx )
      Contact( #EstadoZona.Rearme_CBx )
   END_RUNG wire#w5
   // the same network as SCL:
   "DB1_SalidasExterioresDeMesa".Mesa[#Mesa].Avanzar_E1E3 := (((((#Mx_ET10 AND #AVTF_MEnt) OR #Mx_ET11 OR #Mx_ET12) AND NOT #CNT_pHsMx.QD AND #Selec_M1M2_Entrada) OR ((#Mx_ET02 OR #Mx_ET50 OR #Mx_ET51) AND #PTF_MSal AND #AVTF_MSal AND #Selec_M3M4_Salida)) AND ((#Selec_DW AND #MELEV_DW) OR (#Selec_UP AND #MELEV_UP)) AND #EstadoZona.Marcha_CBx AND NOT #EstadoVI.Error_Mx AND NOT #Error_Tx) OR (NOT #Termico_Tx AND #EstadoZona.Rearme_CBx);
END_REGION

REGION Network 76: SALIDAS - Retroceso E1E3
   RUNG wire#powerrail
      Contact( #Mx_ET10 )
      Contact( #AVTF_MEnt )
      wire#w1
      I_Contact( #CNT_pHsMx.QD )
      Contact( #Selec_M3M4_Entrada )
      wire#w2
      Contact( #Selec_DW )
      Contact( #MELEV_DW )
      wire#w4
      Contact( #EstadoZona.Marcha_CBx )
      I_Contact( #EstadoVI.Error_Mx )
      I_Contact( #Error_Tx )
      wire#w5
      Coil( "DB1_SalidasExterioresDeMesa".Mesa[#Mesa].Retroceder_E1E3 )
   END_RUNG
   RUNG wire#powerrail
      Contact( #Mx_ET11 )
   END_RUNG wire#w1
   RUNG wire#powerrail
      Contact( #Mx_ET12 )
   END_RUNG wire#w1
   RUNG wire#powerrail
      Contact( #Mx_ET02 )
      wire#w3
      Contact( #PTF_MSal )
      Contact( #AVTF_MSal )
      Contact( #Selec_M1M2_Salida )
   END_RUNG wire#w2
   RUNG wire#powerrail
      Contact( #Mx_ET50 )
   END_RUNG wire#w3
   RUNG wire#powerrail
      Contact( #Mx_ET51 )
   END_RUNG wire#w3
   RUNG wire#w2
      Contact( #Selec_UP )
      Contact( #MELEV_UP )
   END_RUNG wire#w4
   RUNG wire#powerrail
      I_Contact( #Termico_Tx )
      Contact( #EstadoZona.Rearme_CBx )
   END_RUNG wire#w5
   // the same network as SCL:
   "DB1_SalidasExterioresDeMesa".Mesa[#Mesa].Retroceder_E1E3 := (((((#Mx_ET10 AND #AVTF_MEnt) OR #Mx_ET11 OR #Mx_ET12) AND NOT #CNT_pHsMx.QD AND #Selec_M3M4_Entrada) OR ((#Mx_ET02 OR #Mx_ET50 OR #Mx_ET51) AND #PTF_MSal AND #AVTF_MSal AND #Selec_M1M2_Salida)) AND ((#Selec_DW AND #MELEV_DW) OR (#Selec_UP AND #MELEV_UP)) AND #EstadoZona.Marcha_CBx AND NOT #EstadoVI.Error_Mx AND NOT #Error_Tx) OR (NOT #Termico_Tx AND #EstadoZona.Rearme_CBx);
END_REGION

REGION Network 77: SALIDAS - Parar E1E3
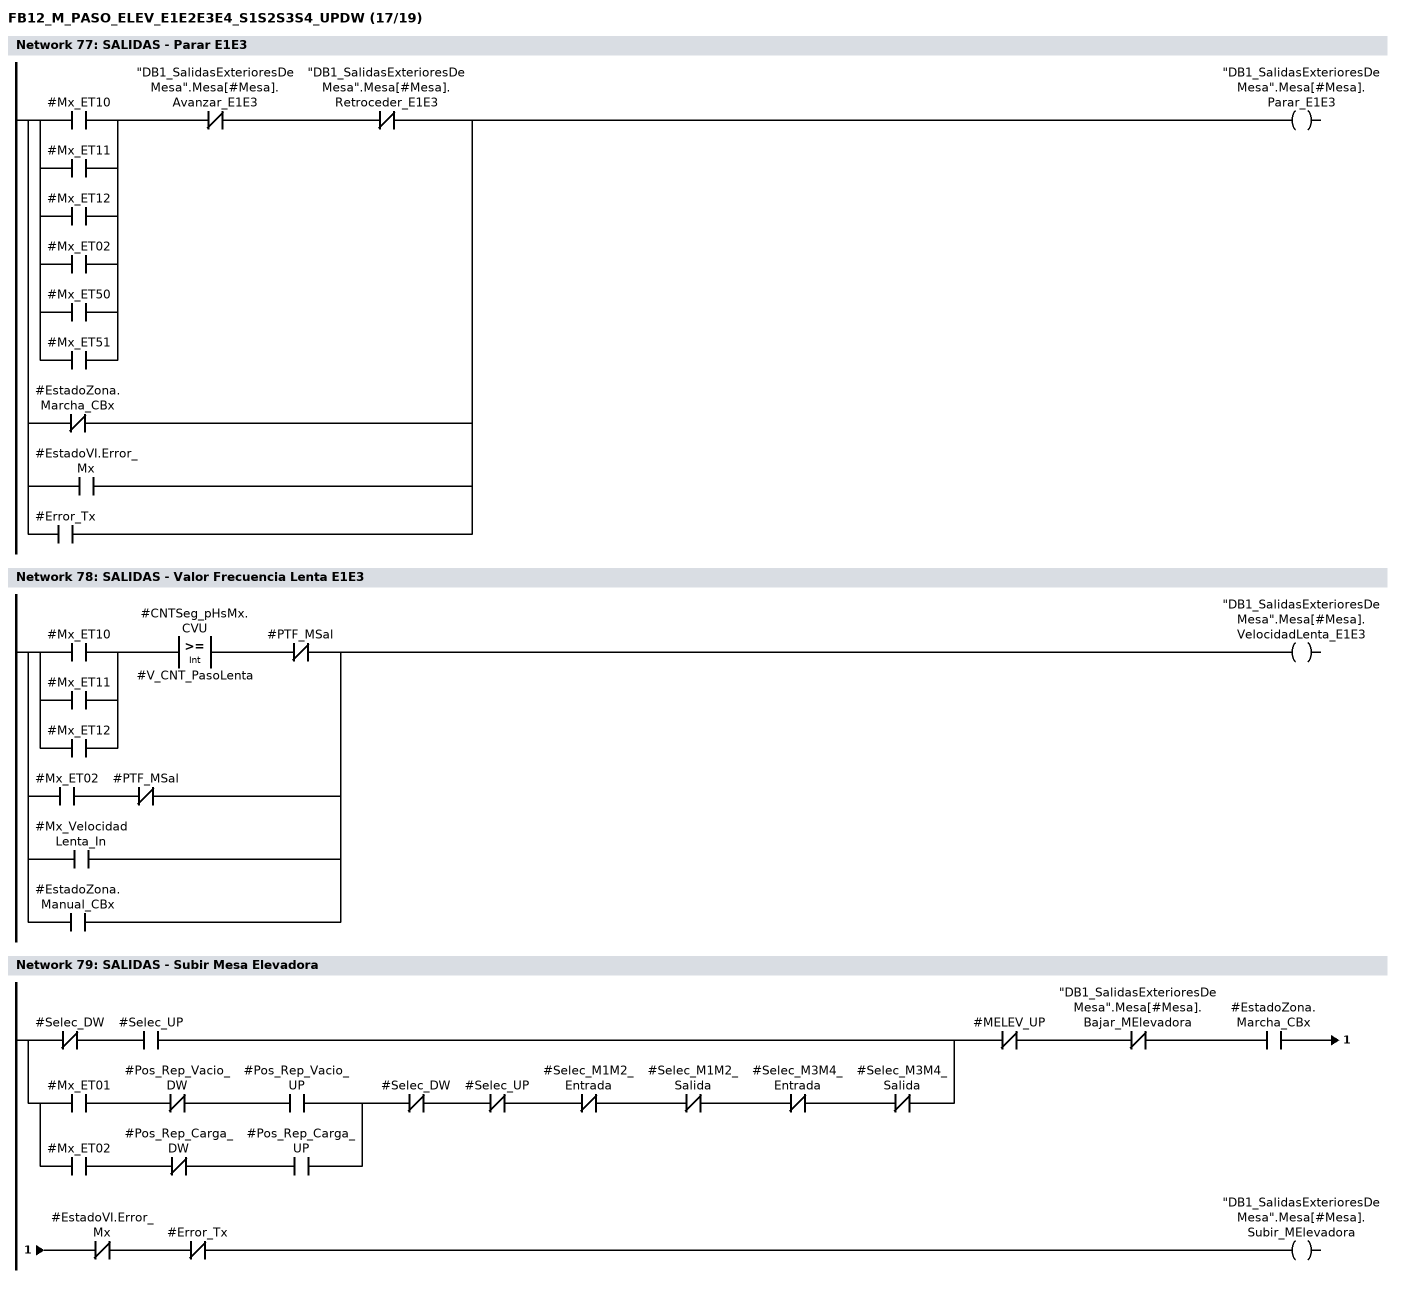
   RUNG wire#powerrail
      Contact( #Mx_ET10 )
      wire#w1
      I_Contact( "DB1_SalidasExterioresDeMesa".Mesa[#Mesa].Avanzar_E1E3 )
      I_Contact( "DB1_SalidasExterioresDeMesa".Mesa[#Mesa].Retroceder_E1E3 )
      wire#w2
      Coil( "DB1_SalidasExterioresDeMesa".Mesa[#Mesa].Parar_E1E3 )
   END_RUNG
   RUNG wire#powerrail
      Contact( #Mx_ET11 )
   END_RUNG wire#w1
   RUNG wire#powerrail
      Contact( #Mx_ET12 )
   END_RUNG wire#w1
   RUNG wire#powerrail
      Contact( #Mx_ET02 )
   END_RUNG wire#w1
   RUNG wire#powerrail
      Contact( #Mx_ET50 )
   END_RUNG wire#w1
   RUNG wire#powerrail
      Contact( #Mx_ET51 )
   END_RUNG wire#w1
   RUNG wire#powerrail
      I_Contact( #EstadoZona.Marcha_CBx )
   END_RUNG wire#w2
   RUNG wire#powerrail
      Contact( #EstadoVI.Error_Mx )
   END_RUNG wire#w2
   RUNG wire#powerrail
      Contact( #Error_Tx )
   END_RUNG wire#w2
   // the same network as SCL:
   "DB1_SalidasExterioresDeMesa".Mesa[#Mesa].Parar_E1E3 := ((#Mx_ET10 OR #Mx_ET11 OR #Mx_ET12 OR #Mx_ET02 OR #Mx_ET50 OR #Mx_ET51) AND NOT "DB1_SalidasExterioresDeMesa".Mesa[#Mesa].Avanzar_E1E3 AND NOT "DB1_SalidasExterioresDeMesa".Mesa[#Mesa].Retroceder_E1E3) OR NOT #EstadoZona.Marcha_CBx OR #EstadoVI.Error_Mx OR #Error_Tx;
END_REGION

REGION Network 78: SALIDAS - Valor Frecuencia Lenta E1E3
   RUNG wire#powerrail
      Contact( #Mx_ET10 )
      wire#w1
      { S7_Templates := "SrcType := Int" } GE_Contact(in1 := #CNTSeg_pHsMx.CVU, in2 := #V_CNT_PasoLenta)
      I_Contact( #PTF_MSal )
      wire#w2
      Coil( "DB1_SalidasExterioresDeMesa".Mesa[#Mesa].VelocidadLenta_E1E3 )
   END_RUNG
   RUNG wire#powerrail
      Contact( #Mx_ET11 )
   END_RUNG wire#w1
   RUNG wire#powerrail
      Contact( #Mx_ET12 )
   END_RUNG wire#w1
   RUNG wire#powerrail
      Contact( #Mx_ET02 )
      I_Contact( #PTF_MSal )
   END_RUNG wire#w2
   RUNG wire#powerrail
      Contact( #Mx_VelocidadLenta_In )
   END_RUNG wire#w2
   RUNG wire#powerrail
      Contact( #EstadoZona.Manual_CBx )
   END_RUNG wire#w2
   // the same network as SCL:
   "DB1_SalidasExterioresDeMesa".Mesa[#Mesa].VelocidadLenta_E1E3 := ((#Mx_ET10 OR #Mx_ET11 OR #Mx_ET12) AND (#CNTSeg_pHsMx.CVU >= #V_CNT_PasoLenta) AND NOT #PTF_MSal) OR (#Mx_ET02 AND NOT #PTF_MSal) OR #Mx_VelocidadLenta_In OR #EstadoZona.Manual_CBx;
END_REGION

REGION Network 79: SALIDAS - Subir Mesa Elevadora
   RUNG wire#powerrail
      I_Contact( #Selec_DW )
      Contact( #Selec_UP )
      wire#w1
      I_Contact( #MELEV_UP )
      I_Contact( "DB1_SalidasExterioresDeMesa".Mesa[#Mesa].Bajar_MElevadora )
      Contact( #EstadoZona.Marcha_CBx )
      I_Contact( #EstadoVI.Error_Mx )
      I_Contact( #Error_Tx )
      Coil( "DB1_SalidasExterioresDeMesa".Mesa[#Mesa].Subir_MElevadora )
   END_RUNG
   RUNG wire#powerrail
      Contact( #Mx_ET01 )
      I_Contact( #Pos_Rep_Vacio_DW )
      Contact( #Pos_Rep_Vacio_UP )
      wire#w2
      I_Contact( #Selec_DW )
      I_Contact( #Selec_UP )
      I_Contact( #Selec_M1M2_Entrada )
      I_Contact( #Selec_M1M2_Salida )
      I_Contact( #Selec_M3M4_Entrada )
      I_Contact( #Selec_M3M4_Salida )
   END_RUNG wire#w1
   RUNG wire#powerrail
      Contact( #Mx_ET02 )
      I_Contact( #Pos_Rep_Carga_DW )
      Contact( #Pos_Rep_Carga_UP )
   END_RUNG wire#w2
   // the same network as SCL:
   "DB1_SalidasExterioresDeMesa".Mesa[#Mesa].Subir_MElevadora := ((NOT #Selec_DW AND #Selec_UP) OR (((#Mx_ET01 AND NOT #Pos_Rep_Vacio_DW AND #Pos_Rep_Vacio_UP) OR (#Mx_ET02 AND NOT #Pos_Rep_Carga_DW AND #Pos_Rep_Carga_UP)) AND NOT #Selec_DW AND NOT #Selec_UP AND NOT #Selec_M1M2_Entrada AND NOT #Selec_M1M2_Salida AND NOT #Selec_M3M4_Entrada AND NOT #Selec_M3M4_Salida)) AND NOT #MELEV_UP AND NOT "DB1_SalidasExterioresDeMesa".Mesa[#Mesa].Bajar_MElevadora AND #EstadoZona.Marcha_CBx AND NOT #EstadoVI.Error_Mx AND NOT #Error_Tx;
END_REGION

REGION Network 80: SALIDAS - Bajar Mesa Elevadora
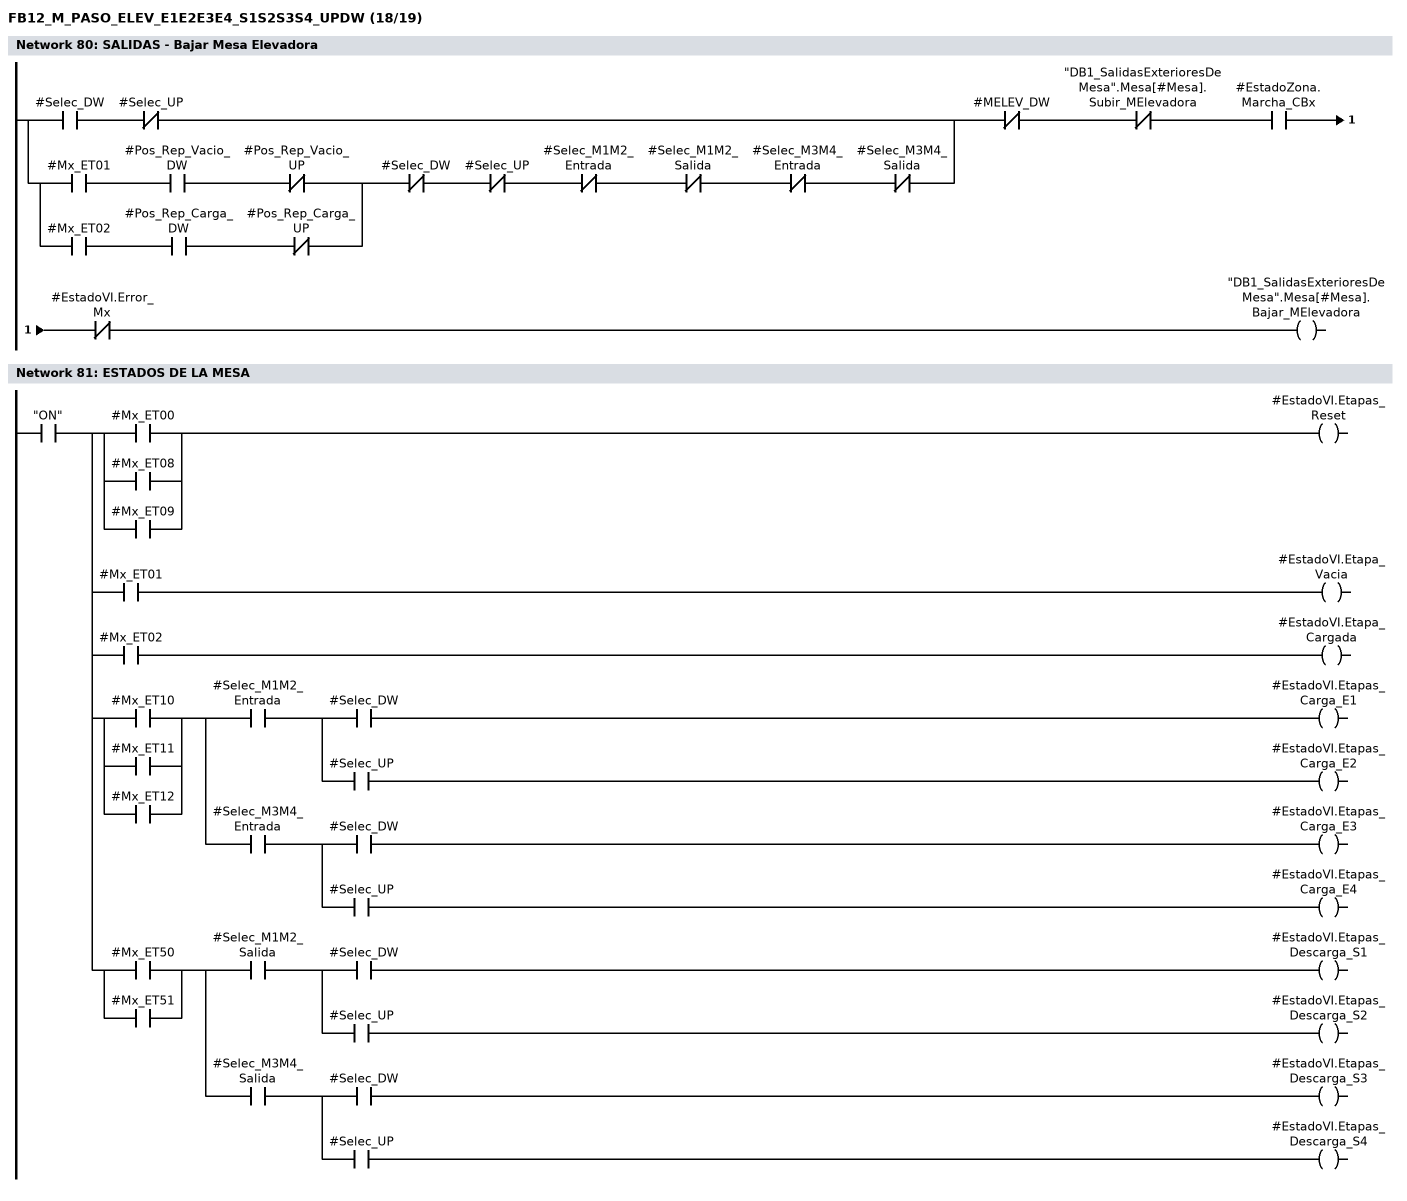
   RUNG wire#powerrail
      Contact( #Selec_DW )
      I_Contact( #Selec_UP )
      wire#w1
      I_Contact( #MELEV_DW )
      I_Contact( "DB1_SalidasExterioresDeMesa".Mesa[#Mesa].Subir_MElevadora )
      Contact( #EstadoZona.Marcha_CBx )
      I_Contact( #EstadoVI.Error_Mx )
      Coil( "DB1_SalidasExterioresDeMesa".Mesa[#Mesa].Bajar_MElevadora )
   END_RUNG
   RUNG wire#powerrail
      Contact( #Mx_ET01 )
      Contact( #Pos_Rep_Vacio_DW )
      I_Contact( #Pos_Rep_Vacio_UP )
      wire#w2
      I_Contact( #Selec_DW )
      I_Contact( #Selec_UP )
      I_Contact( #Selec_M1M2_Entrada )
      I_Contact( #Selec_M1M2_Salida )
      I_Contact( #Selec_M3M4_Entrada )
      I_Contact( #Selec_M3M4_Salida )
   END_RUNG wire#w1
   RUNG wire#powerrail
      Contact( #Mx_ET02 )
      Contact( #Pos_Rep_Carga_DW )
      I_Contact( #Pos_Rep_Carga_UP )
   END_RUNG wire#w2
   // the same network as SCL:
   "DB1_SalidasExterioresDeMesa".Mesa[#Mesa].Bajar_MElevadora := ((#Selec_DW AND NOT #Selec_UP) OR (((#Mx_ET01 AND #Pos_Rep_Vacio_DW AND NOT #Pos_Rep_Vacio_UP) OR (#Mx_ET02 AND #Pos_Rep_Carga_DW AND NOT #Pos_Rep_Carga_UP)) AND NOT #Selec_DW AND NOT #Selec_UP AND NOT #Selec_M1M2_Entrada AND NOT #Selec_M1M2_Salida AND NOT #Selec_M3M4_Entrada AND NOT #Selec_M3M4_Salida)) AND NOT #MELEV_DW AND NOT "DB1_SalidasExterioresDeMesa".Mesa[#Mesa].Subir_MElevadora AND #EstadoZona.Marcha_CBx AND NOT #EstadoVI.Error_Mx;
END_REGION

REGION Network 81: ESTADOS DE LA MESA
   RUNG wire#powerrail
      Contact( "ON" )
      wire#w1
      Contact( #Mx_ET00 )
      wire#w2
      Coil( #EstadoVI.Etapas_Reset )
   END_RUNG
   RUNG wire#w1
      Contact( #Mx_ET08 )
   END_RUNG wire#w2
   RUNG wire#w1
      Contact( #Mx_ET09 )
   END_RUNG wire#w2
   RUNG wire#w1
      Contact( #Mx_ET01 )
      Coil( #EstadoVI.Etapa_Vacia )
   END_RUNG
   RUNG wire#w1
      Contact( #Mx_ET02 )
      Coil( #EstadoVI.Etapa_Cargada )
   END_RUNG
   RUNG wire#w1
      Contact( #Mx_ET10 )
      wire#w3
      Contact( #Selec_M1M2_Entrada )
      wire#w4
      Contact( #Selec_DW )
      Coil( #EstadoVI.Etapas_Carga_E1 )
   END_RUNG
   RUNG wire#w1
      Contact( #Mx_ET11 )
   END_RUNG wire#w3
   RUNG wire#w1
      Contact( #Mx_ET12 )
   END_RUNG wire#w3
   RUNG wire#w4
      Contact( #Selec_UP )
      Coil( #EstadoVI.Etapas_Carga_E2 )
   END_RUNG
   RUNG wire#w3
      Contact( #Selec_M3M4_Entrada )
      wire#w5
      Contact( #Selec_DW )
      Coil( #EstadoVI.Etapas_Carga_E3 )
   END_RUNG
   RUNG wire#w5
      Contact( #Selec_UP )
      Coil( #EstadoVI.Etapas_Carga_E4 )
   END_RUNG
   RUNG wire#w1
      Contact( #Mx_ET50 )
      wire#w6
      Contact( #Selec_M1M2_Salida )
      wire#w7
      Contact( #Selec_DW )
      Coil( #EstadoVI.Etapas_Descarga_S1 )
   END_RUNG
   RUNG wire#w1
      Contact( #Mx_ET51 )
   END_RUNG wire#w6
   RUNG wire#w7
      Contact( #Selec_UP )
      Coil( #EstadoVI.Etapas_Descarga_S2 )
   END_RUNG
   RUNG wire#w6
      Contact( #Selec_M3M4_Salida )
      wire#w8
      Contact( #Selec_DW )
      Coil( #EstadoVI.Etapas_Descarga_S3 )
   END_RUNG
   RUNG wire#w8
      Contact( #Selec_UP )
      Coil( #EstadoVI.Etapas_Descarga_S4 )
   END_RUNG
   // the same network as SCL:
   #EstadoVI.Etapas_Reset := "ON" AND (#Mx_ET00 OR #Mx_ET08 OR #Mx_ET09);
   #EstadoVI.Etapa_Vacia := "ON" AND #Mx_ET01;
   #EstadoVI.Etapa_Cargada := "ON" AND #Mx_ET02;
   #_w1 := "ON" AND (#Mx_ET10 OR #Mx_ET11 OR #Mx_ET12);
   #_w2 := #_w1 AND #Selec_M1M2_Entrada;
   #EstadoVI.Etapas_Carga_E1 := #_w2 AND #Selec_DW;
   #EstadoVI.Etapas_Carga_E2 := #_w2 AND #Selec_UP;
   #_w3 := #_w1 AND #Selec_M3M4_Entrada;
   #EstadoVI.Etapas_Carga_E3 := #_w3 AND #Selec_DW;
   #EstadoVI.Etapas_Carga_E4 := #_w3 AND #Selec_UP;
   #_w4 := "ON" AND (#Mx_ET50 OR #Mx_ET51);
   #_w5 := #_w4 AND #Selec_M1M2_Salida;
   #EstadoVI.Etapas_Descarga_S1 := #_w5 AND #Selec_DW;
   #EstadoVI.Etapas_Descarga_S2 := #_w5 AND #Selec_UP;
   #_w6 := #_w4 AND #Selec_M3M4_Salida;
   #EstadoVI.Etapas_Descarga_S3 := #_w6 AND #Selec_DW;
   #EstadoVI.Etapas_Descarga_S4 := #_w6 AND #Selec_UP;
END_REGION

REGION Network 82: ENTRADAS DE LA MESA
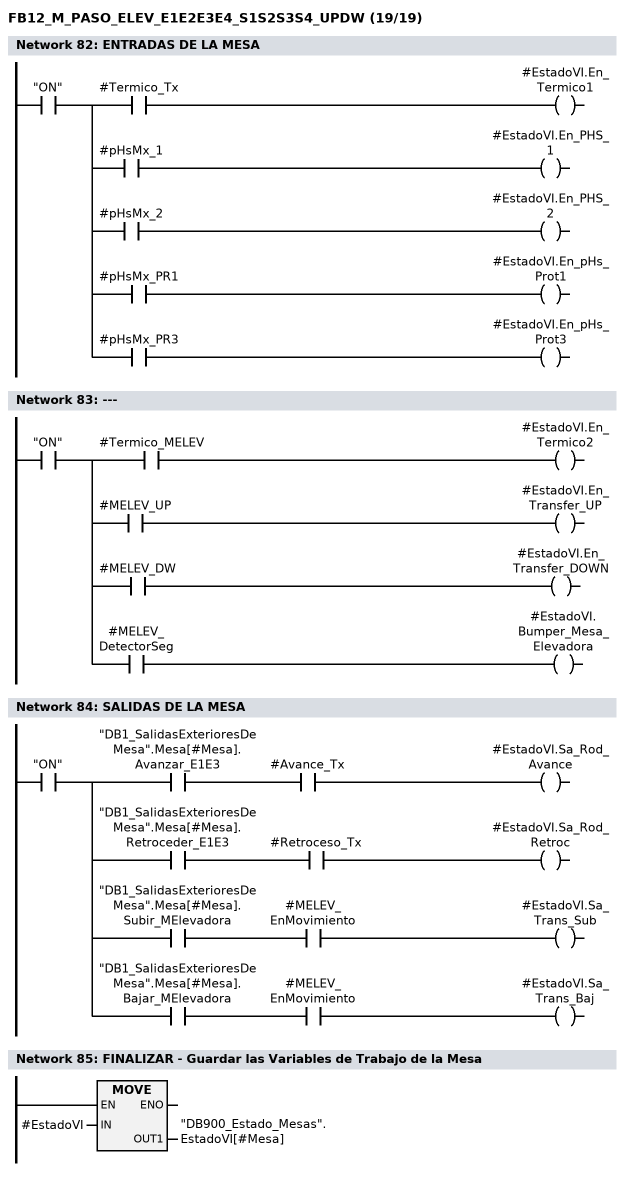
   RUNG wire#powerrail
      Contact( "ON" )
      wire#w1
      Contact( #Termico_Tx )
      Coil( #EstadoVI.En_Termico1 )
   END_RUNG
   RUNG wire#w1
      Contact( #pHsMx_1 )
      Coil( #EstadoVI.En_PHS_1 )
   END_RUNG
   RUNG wire#w1
      Contact( #pHsMx_2 )
      Coil( #EstadoVI.En_PHS_2 )
   END_RUNG
   RUNG wire#w1
      Contact( #pHsMx_PR1 )
      Coil( #EstadoVI.En_pHs_Prot1 )
   END_RUNG
   RUNG wire#w1
      Contact( #pHsMx_PR3 )
      Coil( #EstadoVI.En_pHs_Prot3 )
   END_RUNG
   // the same network as SCL:
   #EstadoVI.En_Termico1 := "ON" AND #Termico_Tx;
   #EstadoVI.En_PHS_1 := "ON" AND #pHsMx_1;
   #EstadoVI.En_PHS_2 := "ON" AND #pHsMx_2;
   #EstadoVI.En_pHs_Prot1 := "ON" AND #pHsMx_PR1;
   #EstadoVI.En_pHs_Prot3 := "ON" AND #pHsMx_PR3;
END_REGION

REGION Network 83: ---
   RUNG wire#powerrail
      Contact( "ON" )
      wire#w1
      Contact( #Termico_MELEV )
      Coil( #EstadoVI.En_Termico2 )
   END_RUNG
   RUNG wire#w1
      Contact( #MELEV_UP )
      Coil( #EstadoVI.En_Transfer_UP )
   END_RUNG
   RUNG wire#w1
      Contact( #MELEV_DW )
      Coil( #EstadoVI.En_Transfer_DOWN )
   END_RUNG
   RUNG wire#w1
      Contact( #MELEV_DetectorSeg )
      Coil( #EstadoVI.Bumper_Mesa_Elevadora )
   END_RUNG
   // the same network as SCL:
   #EstadoVI.En_Termico2 := "ON" AND #Termico_MELEV;
   #EstadoVI.En_Transfer_UP := "ON" AND #MELEV_UP;
   #EstadoVI.En_Transfer_DOWN := "ON" AND #MELEV_DW;
   #EstadoVI.Bumper_Mesa_Elevadora := "ON" AND #MELEV_DetectorSeg;
END_REGION

REGION Network 84: SALIDAS DE LA MESA
   RUNG wire#powerrail
      Contact( "ON" )
      wire#w1
      Contact( "DB1_SalidasExterioresDeMesa".Mesa[#Mesa].Avanzar_E1E3 )
      Contact( #Avance_Tx )
      Coil( #EstadoVI.Sa_Rod_Avance )
   END_RUNG
   RUNG wire#w1
      Contact( "DB1_SalidasExterioresDeMesa".Mesa[#Mesa].Retroceder_E1E3 )
      Contact( #Retroceso_Tx )
      Coil( #EstadoVI.Sa_Rod_Retroc )
   END_RUNG
   RUNG wire#w1
      Contact( "DB1_SalidasExterioresDeMesa".Mesa[#Mesa].Subir_MElevadora )
      Contact( #MELEV_EnMovimiento )
      Coil( #EstadoVI.Sa_Trans_Sub )
   END_RUNG
   RUNG wire#w1
      Contact( "DB1_SalidasExterioresDeMesa".Mesa[#Mesa].Bajar_MElevadora )
      Contact( #MELEV_EnMovimiento )
      Coil( #EstadoVI.Sa_Trans_Baj )
   END_RUNG
   // the same network as SCL:
   #EstadoVI.Sa_Rod_Avance := "ON" AND "DB1_SalidasExterioresDeMesa".Mesa[#Mesa].Avanzar_E1E3 AND #Avance_Tx;
   #EstadoVI.Sa_Rod_Retroc := "ON" AND "DB1_SalidasExterioresDeMesa".Mesa[#Mesa].Retroceder_E1E3 AND #Retroceso_Tx;
   #EstadoVI.Sa_Trans_Sub := "ON" AND "DB1_SalidasExterioresDeMesa".Mesa[#Mesa].Subir_MElevadora AND #MELEV_EnMovimiento;
   #EstadoVI.Sa_Trans_Baj := "ON" AND "DB1_SalidasExterioresDeMesa".Mesa[#Mesa].Bajar_MElevadora AND #MELEV_EnMovimiento;
END_REGION

REGION Network 85: FINALIZAR - Guardar las Variables de Trabajo de la Mesa
   RUNG wire#powerrail
      Move(in := #EstadoVI, out1 => "DB900_Estado_Mesas".EstadoVI[#Mesa])
   END_RUNG
   // the same network as SCL:
   "DB900_Estado_Mesas".EstadoVI[#Mesa] := #EstadoVI;
END_REGION
END_FUNCTION_BLOCK
